VAR_IN_OUT
	rBnt_BlueflagNum: UINT;
	rBnt_Blueflaging: BOOL;	
	NumberPos: ARRAY[0..20] OF LREAL;//接带点记录数据
	NumberPos1: ARRAY[0..20] OF LREAL;//接带点记录数据
	NumberPos2: ARRAY[0..20] OF LREAL;//接带点记录数据
END_VAR

rBnt_Blueflag(CLK:=Bnt_Blueflag , Q=> );	// 接带输入信号
rFlagDone(CLK:=FlagDone , Q=> );	// 电芯下料完成信号
//根据接带信号记录放卷轴当前的角度
IF rBnt_Blueflag.Q THEN
		rBnt_Blueflaging:=TRUE;//接带信号
		rBnt_BlueflagNum:=rBnt_BlueflagCaNum;
		FOR i:=0 TO 20 BY 1 DO
							IF i<20 THEN
									NumberPos[20-i]:=	NumberPos[19-i];
							ELSE
									NumberPos[0]:=AixsoActPos;
							END_IF;
							
							IF i<20 THEN
									NumberPos1[20-i]:=	NumberPos1[19-i];
							ELSE
									NumberPos1[0]:=AixsoActPos+fYDLength;
							END_IF;
							
							IF i<20 THEN
									NumberPos2[20-i]:=	NumberPos2[19-i];
							ELSE
									NumberPos2[0]:=AixsoActPos+fYDLength*2;
							END_IF;
		END_FOR
END_IF
//根据当前的角度
FOR i:=0 TO 20 BY 1 DO
		IF NumberPos[i]<>0 THEN
			RemberPos[i]:= FC_AngleToLength(ABS(AixsoActPos-NumberPos[i]),Diameter);			
		END_IF
		
		IF NumberPos1[i]<>0 THEN
			RemberPos1[i]:= FC_AngleToLength(ABS(AixsoActPos-NumberPos1[i]),Diameter);
		END_IF
		
		IF NumberPos2[i]<>0 THEN
			RemberPos2[i]:= FC_AngleToLength(ABS(AixsoActPos-NumberPos2[i]),Diameter);
		END_IF

		IF (RemberPos[i] >= SetLenght AND NumberPos[i]<>0) OR (RemberPos1[i] >= SetLenght AND NumberPos1[i]<>0)OR (RemberPos2[i] >= SetLenght AND NumberPos2[i]<>0)   THEN
			FlagPoisn[i]:=TRUE;
		END_IF
		
		IF (RemberPos[i] >= SetLenght AND NumberPos[i]<>0) AND rFlagDone.Q THEN
			FlagPoisn[i] :=FALSE;
			NumberPos[i]:=0;
		END_IF
	
		IF (RemberPos1[i] >= SetLenght AND NumberPos1[i]<>0) AND rFlagDone.Q THEN
			FlagPoisn[i] :=FALSE;
			NumberPos1[i]:=0;
		END_IF	

		IF (RemberPos2[i] >= SetLenght AND NumberPos2[i]<>0) AND rFlagDone.Q THEN
			FlagPoisn[i] :=FALSE;
			NumberPos2[i]:=0;
		END_IF		
END_FOR

END_FUNCTION_BLOCK

// ---- P2POUs/BasicFunction/09_User1/FB_CrectCamUpDown_4.TcPOU
FUNCTION_BLOCK FB_CrectCamUpDown_4	
VAR_INPUT
   	bCreatTable		                         :BOOL;	
	Reset                                        :BOOL;  
	iTable		                                :UINT;    

	fInitLength									:REAL;//耦合的初始高度
    fMoveLength                              :REAL;   //目标取或放料高度
    fSaveLength                               :REAL;    //升降安全高度

    fMasterKeyPos1                           :REAL:=208;   
    fMasterKeyPos2                           :REAL:=256;   
END_VAR

VAR_IN_OUT
	axisSlave		                            :axis_ref;  
	axisMaster		                            :axis_ref;  
END_VAR

VAR_OUTPUT
    bCreatTableDone                        :BOOL;
    bCreatTableError                        :BOOL;
	bError                         :BOOL;

END_VAR


VAR
	rtrigs		                                      :ARRAY[1..3]OF R_TRIG;
	ftrigs		                                      :ARRAY[1..3]OF F_TRIG;
    PositionData1			                  :ARRAY[1..8] OF MC_MotionFunctionPoint;	////
	fbCamtableselect:		               	MC_CamTableSelect;////
	Cam_table:				MC_CAM_REF;////
	bWriteCamData: BOOL;
    iCreatTableStep       :INT;
END_VAR


rtrigs[1](CLK:=bCreatTable);  
ftrigs[1](CLK:=bCreatTable);  

CASE iCreatTableStep OF   
0:  
    IF  rtrigs[1].Q  AND NOT bCreatTableError  THEN
         fbCamtableselect.Execute:=FALSE;
         bCreatTableDone:=FALSE;
         bCreatTable:=FALSE;
         bWriteCamData:=TRUE;
         iCreatTableStep:=10;
    END_IF 

10: 
   IF NOT bWriteCamData THEN 
	  fbCamtableselect.Execute:=TRUE;   
	 iCreatTableStep:=20;	
  END_IF

20:		
	IF NOT  fbCamtableselect.Execute   THEN
        bCreatTableDone:=TRUE;
		iCreatTableStep:=0;	
    ELSIF  fbCamtableselect.Error        THEN
       bCreatTableError:=TRUE;
       iCreatTableStep:=999;	//创建凸轮失败
	END_IF		
END_CASE

(**********故障***********)
	IF  Reset  AND bCreatTableError  THEN  
	   bCreatTableError:=FALSE;
	   iCreatTableStep:=0;
	END_IF


ModifyCam();

ACTION ModifyCam:

fbCamtableselect(   
	Execute:=                        fbCamtableselect.Execute ,
	Periodic:=                        FALSE ,
	MasterAbsolute:=             FALSE,
	SlaveAbsolute:=                FALSE ,
	CamTableID:=                  iTable,
	Master:=                         axisMaster ,
	Slave:=                            axisSlave ,
	CamTable:=                     Cam_table , );

IF fbCamtableselect.Done THEN
    fbCamtableselect.Execute:=FALSE;
END_IF

IF bWriteCamData  THEN
 
	  Cam_table.ArraySize:=SIZEOF(PositionData1); 
	  Cam_table.NoOfColumns:=1;
	  Cam_table.NoOfRows:=4;
	  Cam_table.pArray:=ADR(PositionData1);
	  Cam_table.TableType:=MC_TABLETYPE_MOTIONFUNCTION;
  
      //MOTIONFUNCTYPE_BESCHLTRAPEZ     MOTIONFUNCTYPE_POLYNOM7_MM    MOTIONFUNCTYPE_BESCHLTRAPEZ   MOTIONFUNCTYPE_POLYNOM1

	  PositionData1[1].	PointIndex	:=	        1;
	  PositionData1[1].	FunctionType	:=		MOTIONFUNCTYPE_POLYNOM5_MM;//MOTIONFUNCTYPE_BESCHLTRAPEZ     MOTIONFUNCTYPE_POLYNOM7_MM    MOTIONFUNCTYPE_BESCHLTRAPEZ
	  PositionData1[1].	PointType	:=	        MOTIONPOINTTYPE_MOTION;
	  PositionData1[1].	RelIndexNextPoint	:=  1;
	  PositionData1[1].	MasterPos	:=	        0;
	  PositionData1[1].	SlavePos	:=	        0;		//fMoveLength
	  PositionData1[1].	SlaveVelo	:=	        0;
	  
	  PositionData1[2].	PointIndex	:=	        2;
	  PositionData1[2].	FunctionType	:=		MOTIONFUNCTYPE_POLYNOM5_MM;
	  PositionData1[2].	PointType	:=	        MOTIONPOINTTYPE_MOTION;
	  PositionData1[2].	RelIndexNextPoint	:=  1;
	  PositionData1[2].	MasterPos	:=	        fMasterKeyPos1;//fMasterKeyPos
	  PositionData1[2].	SlavePos	:=	        fSaveLength - fInitLength;	
	  PositionData1[2].	SlaveVelo	:=	        0;//(fInitLength-fSaveLength)/fMasterKeyPos1	;

	  PositionData1[3].	PointIndex	:=	        3;//SJ
	  PositionData1[3].	FunctionType	:=		MOTIONFUNCTYPE_POLYNOM1;
	  PositionData1[3].	PointType	:=	        MOTIONPOINTTYPE_MOTION;
	  PositionData1[3].	RelIndexNextPoint	:=  1;
	  PositionData1[3].	MasterPos	:=	        fMasterKeyPos2;//fMasterKeyPos
	  PositionData1[3].	SlavePos	:=	        0;	
	  PositionData1[3].	SlaveVelo	:=	        0;//(fInitLength-fSaveLength)/fMasterKeyPos1	;	  
	  
	  
	  PositionData1[4].	PointIndex	:=	        4;
	  PositionData1[4].	FunctionType	:=		MOTIONFUNCTYPE_POLYNOM5_MM;
	  PositionData1[4].	PointType	:=	        MOTIONPOINTTYPE_MOTION;
	  PositionData1[4].	RelIndexNextPoint	:=  0;
	  PositionData1[4].	MasterPos	:=	        360;//fMasterKeyPos
	  PositionData1[4].	SlavePos	:=	        0;	
	  PositionData1[4].	SlaveVelo	:=	        0;//(fInitLength-fSaveLength)/fMasterKeyPos1	;
	  



     bWriteCamData:=FALSE;
END_IF
END_ACTION

END_FUNCTION_BLOCK

// ---- P2POUs/BasicFunction/12_User2/FB_DiameterORLength.TcPOU
FUNCTION_BLOCK FB_DiameterORLength
VAR_INPUT
	D1 : REAL; //外直径
	R1 : REAL:=172; //内直径
	T1 : REAL; //隔膜厚度
END_VAR
VAR_OUTPUT
	OUT1: REAL;
END_VAR
VAR
	R2: REAL;
	R3: REAL;
	R4: REAL;
	
END_VAR

IF  T1 <> 0 AND D1 >= R1 THEN
	R2:=(D1-R1)/2  ;  
	R3:=((D1*Tc2_System.PI)+(R1*Tc2_System.PI))/2 ;  //平均长度
	R4:=R2/T1;  //总层数
	OUT1:=(R4*R3)/1000;
END_IF

END_FUNCTION_BLOCK

// ---- P2POUs/BasicFunction/12_User2/FB_RectifyTry.TcPOU
FUNCTION_BLOCK FB_RectifyTry
VAR_INPUT
	Execute: BOOL;// 测试启动HMI
	AxisNO_X: INT; // X轴	
	AxisNO_Y: INT; // Y轴	
	AxisNO_R: INT; // R轴	
	Demarcate_X:REAL;//X轴纠偏位
	Demarcate_Y:REAL;//Y轴纠偏位	
	Demarcate_R:REAL;//R轴纠偏位		
	// CCD拍照记录次数
	CCDNo: INT;
END_VAR
VAR_OUTPUT
END_VAR
VAR
	Step0: INT;
	r_TRIG: R_TRIG;

	// 延时复位CCD拍照启动
	TON1: TON;
	TON2: TON;
	i: INT;
END_VAR

VAR_IN_OUT
	// 启动CCD拍照
	CCDStart: BOOL;
END_VAR

//纠偏平台定位精度数据测试
r_TRIG(CLK:=Execute , Q=> );
TON1(IN:= , PT:=T#2S , Q=> , ET=> );
TON2(IN:= , PT:=T#0.3S , Q=> , ET=> );

CASE Step0 OF
	0://判断是否启动测试
		IF r_TRIG.Q THEN
			i:=0;
			Step0:=10;
			TON2.IN:=FALSE;
		END_IF
	10://纠偏平台X、Y回初始位
		IF arrAxisCtrl[AxisNO_X].Status.Homed AND arrAxisCtrl[AxisNO_X].Status.NoMoving THEN
				IF arrAxisCtrl[AxisNO_X].Cmd.arrbRealPoint[1] THEN
					arrAxisCtrl[AxisNO_X].Cmd.iGoSetPos:=0;
				ELSE
					arrAxisCtrl[AxisNO_X].Cmd.iGoSetPos:=1;
				END_IF
		END_IF
		IF arrAxisCtrl[AxisNO_Y].Status.Homed AND arrAxisCtrl[AxisNO_Y].Status.NoMoving  THEN
				IF arrAxisCtrl[AxisNO_Y].Cmd.arrbRealPoint[1] THEN
					arrAxisCtrl[AxisNO_Y].Cmd.iGoSetPos:=0;
				ELSE
					arrAxisCtrl[AxisNO_Y].Cmd.iGoSetPos:=1;
				END_IF
		END_IF	
	  IF arrAxisCtrl[AxisNO_R].Status.Homed AND arrAxisCtrl[AxisNO_R].Status.NoMoving  THEN
			IF arrAxisCtrl[AxisNO_R].Cmd.arrbRealPoint[1] THEN
				arrAxisCtrl[AxisNO_R].Cmd.iGoSetPos:=0;							       
			ELSE
				arrAxisCtrl[AxisNO_R].Cmd.iGoSetPos:=1;
			END_IF
		END_IF		
		
		IF  arrAxisCtrl[AxisNO_X].Cmd.arrbRealPoint[1]  AND arrAxisCtrl[AxisNO_Y].Cmd.arrbRealPoint[1]  AND arrAxisCtrl[AxisNO_R].Cmd.arrbRealPoint[1] AND
			 arrAxisCtrl[AxisNO_X].Status.Homed AND  arrAxisCtrl[AxisNO_Y].Status.Homed AND arrAxisCtrl[AxisNO_R].Status.Homed THEN
				Step0:=30;
				TON2.IN:=TRUE;
		END_IF	
	(*20://纠偏平台R回初始位
		IF arrAxisCtrl[AxisNO_R].Status.Homed AND arrAxisCtrl[AxisNO_R].Status.NoMoving  THEN
			IF arrAxisCtrl[AxisNO_R].Cmd.arrbRealPoint[1] THEN
				arrAxisCtrl[AxisNO_R].Cmd.iGoSetPos:=0;
				Step0:=30;									       
			ELSE
				arrAxisCtrl[AxisNO_R].Cmd.iGoSetPos:=1;
			END_IF
		END_IF*)
	30://启动CCD拍照
	  IF TON2.Q THEN
		CCDStart:=TRUE;   //CCD拍照启动
		TON2.IN:=FALSE;
		Step0:=40;
	  END_IF	
	40://延时复位CDD拍照启动信号
		IF NOT TON1.Q THEN
			TON1.IN:=TRUE;
		ELSE
			CCDStart:=FALSE;   //CCD拍照启动
			TON1.IN:=FALSE;
			Step0:=50;
		END_IF
	50://纠偏平台X、Y纠偏量
		arrAxisPar[AxisNO_X].arrTargetPoint[6]:=arrAxisPar[AxisNO_X].arrTargetPoint[1] + Demarcate_X;
		arrAxisPar[AxisNO_Y].arrTargetPoint[6]:=arrAxisPar[AxisNO_Y].arrTargetPoint[1] + Demarcate_Y;
		arrAxisPar[AxisNO_R].arrTargetPoint[6]:=arrAxisPar[AxisNO_R].arrTargetPoint[1] +Demarcate_R;
		Step0:=60;	
		TON2.IN:=FALSE;
	60://纠偏平台X、Y移动至纠偏位
 		IF arrAxisCtrl[AxisNO_X].Status.Homed AND arrAxisCtrl[AxisNO_X].Status.NoMoving THEN
				IF arrAxisCtrl[AxisNO_X].Cmd.arrbRealPoint[6] THEN
					arrAxisCtrl[AxisNO_X].Cmd.iGoSetPos:=0;
				ELSE
					arrAxisCtrl[AxisNO_X].Cmd.iGoSetPos:=6;
				END_IF
		END_IF
		IF arrAxisCtrl[AxisNO_Y].Status.Homed AND arrAxisCtrl[AxisNO_Y].Status.NoMoving  THEN
				IF arrAxisCtrl[AxisNO_Y].Cmd.arrbRealPoint[6] THEN
					arrAxisCtrl[AxisNO_Y].Cmd.iGoSetPos:=0;
				ELSE
					arrAxisCtrl[AxisNO_Y].Cmd.iGoSetPos:=6;
				END_IF
		END_IF	
		
	 	IF arrAxisCtrl[AxisNO_R].Status.Homed AND arrAxisCtrl[AxisNO_R].Status.NoMoving THEN
				IF arrAxisCtrl[AxisNO_R].Cmd.arrbRealPoint[6] THEN
					arrAxisCtrl[AxisNO_R].Cmd.iGoSetPos:=0;
				ELSE
					arrAxisCtrl[AxisNO_R].Cmd.iGoSetPos:=6;
				END_IF
		END_IF
	
		IF  arrAxisCtrl[AxisNO_X].Cmd.arrbRealPoint[6]  AND arrAxisCtrl[AxisNO_Y].Cmd.arrbRealPoint[6] AND arrAxisCtrl[AxisNO_R].Cmd.arrbRealPoint[6]  AND 
			 arrAxisCtrl[AxisNO_X].Status.Homed AND  arrAxisCtrl[AxisNO_Y].Status.Homed AND  arrAxisCtrl[AxisNO_R].Status.Homed  THEN
			 Step0:=90;
			 TON2.IN:=TRUE;
		END_IF	 
	(*	
	70://纠偏平台R纠偏量
		arrAxisPar[AxisNO_R].arrTargetPoint[4]:=arrAxisPar[AxisNO_R].arrTargetPoint[1] +Demarcate_R;//arrAxisPar[AxisNO_R].arrTargetPoint[1] + 80*SIN(DEG_TO_RAD(Demarcate_R)) ;
		Step0:=80;
	80://纠偏平台R移动到纠偏位
 		IF arrAxisCtrl[AxisNO_R].Status.Homed AND arrAxisCtrl[AxisNO_R].Status.NoMoving THEN
				IF arrAxisCtrl[AxisNO_R].Cmd.arrbRealPoint[4] THEN
					arrAxisCtrl[AxisNO_R].Cmd.iGoSetPos:=0;
				ELSE
					arrAxisCtrl[AxisNO_R].Cmd.iGoSetPos:=4;
				END_IF
		END_IF
		IF  arrAxisCtrl[AxisNO_R].Cmd.arrbRealPoint[4]  AND arrAxisCtrl[AxisNO_R].Status.Homed THEN
			 Step0:=90;
		END_IF	 *)
	90://启动CCD拍照
	IF TON2.Q THEN
		CCDStart:=TRUE;   //CCD拍照启动
		i:=i+1;
		Step0:=100;
		 TON2.IN:=FALSE;
	END_IF		
	100://延时复位CDD拍照启动信号
		IF NOT TON1.Q THEN
			TON1.IN:=TRUE;
		ELSE
			CCDStart:=FALSE;   //CCD拍照启动
			TON1.IN:=FALSE;
			Step0:=110;
		END_IF
	110://判断是否达到设定次数
		IF i>=CCDNo THEN
			i:=0;
			Step0:=0;
		ELSE
			Step0:=10;
		END_IF
END_CASE

END_FUNCTION_BLOCK

// ---- P2POUs/BasicFunction/12_User2/FB_SuckerTest.TcPOU
FUNCTION_BLOCK FB_SuckerTest
VAR_INPUT
	Execute: BOOL;// 测试启动HMI
	AxisNO_1: INT; // 升降轴
	AxisNO_2: INT;//平移轴
	AxisNO_X: INT; // X轴	
	AxisNO_Y: INT; // Y轴	
	AxisNO_R: INT; // R轴	
	CCD_X1:REAL;//CCD拍照X轴方向的纠偏值
	CCD_X2:REAL;//CCD拍照Y轴方的纠偏值
	CCD_Y:REAL;//CCD拍照旋转方向的纠偏值	
	DTCarryingVacuum: INT;//叠台真空
	deviationVacuum: INT;//纠偏平台真空
	deviationVacuumBark: INT;//纠偏平台破真空
	CCDCount: INT;//测试次数
	DTiMode: INT;
END_VAR
VAR_OUTPUT
END_VAR
VAR
	Step0: INT;
	i: INT;
	r_TRIG:R_TRIG;
	TON1: TON;
	TON2: TON;
	TON3: TON;
	TON4: TON;
END_VAR
VAR_IN_OUT
	// 启动CCD拍照
	CCDStart: BOOL;
END_VAR

r_TRIG(CLK:=Execute , Q=> );
TON1(IN:= , PT:=T#0.5S , Q=> , ET=> );
TON2(IN:= , PT:=T#0.3S , Q=> , ET=> );
TON3(IN:= , PT:=T#0.3S , Q=> , ET=> );
TON4(IN:= , PT:=T#0.3S , Q=> , ET=> );
IF DTiMode=3 THEN
CASE Step0 OF
	0://判断是否启动测试
		IF r_TRIG.Q THEN
			i:=0;
			Step0:=10;
			TON2.IN:=FALSE;
		END_IF
	10://纠偏平台X、Y、R 回初始位 、叠台升降去等待高度、
	   IF arrAxisCtrl[AxisNO_1].Status.Homed AND arrAxisCtrl[AxisNO_1].Status.NoMoving THEN
				IF arrAxisCtrl[AxisNO_1].Cmd.arrbRealPoint[4] THEN
					arrAxisCtrl[AxisNO_1].Cmd.iGoSetPos:=0;
				ELSE
					arrAxisCtrl[AxisNO_1].Cmd.iGoSetPos:=4;
				END_IF
		END_IF
		
		IF arrAxisCtrl[AxisNO_X].Status.Homed AND arrAxisCtrl[AxisNO_X].Status.NoMoving THEN
				IF arrAxisCtrl[AxisNO_X].Cmd.arrbRealPoint[1] THEN
					arrAxisCtrl[AxisNO_X].Cmd.iGoSetPos:=0;
				ELSE
					arrAxisCtrl[AxisNO_X].Cmd.iGoSetPos:=1;
				END_IF
		END_IF
		IF arrAxisCtrl[AxisNO_Y].Status.Homed AND arrAxisCtrl[AxisNO_Y].Status.NoMoving  THEN
				IF arrAxisCtrl[AxisNO_Y].Cmd.arrbRealPoint[1] THEN
					arrAxisCtrl[AxisNO_Y].Cmd.iGoSetPos:=0;
				ELSE
					arrAxisCtrl[AxisNO_Y].Cmd.iGoSetPos:=1;
				END_IF
		END_IF	
	  IF arrAxisCtrl[AxisNO_R].Status.Homed AND arrAxisCtrl[AxisNO_R].Status.NoMoving  THEN
			IF arrAxisCtrl[AxisNO_R].Cmd.arrbRealPoint[1] THEN
				arrAxisCtrl[AxisNO_R].Cmd.iGoSetPos:=0;							       
			ELSE
				arrAxisCtrl[AxisNO_R].Cmd.iGoSetPos:=1;
			END_IF
		END_IF		
		
		IF  arrAxisCtrl[AxisNO_X].Cmd.arrbRealPoint[1]  AND arrAxisCtrl[AxisNO_Y].Cmd.arrbRealPoint[1]  AND arrAxisCtrl[AxisNO_R].Cmd.arrbRealPoint[1] AND
		    arrAxisCtrl[AxisNO_1].Status.NoMoving AND arrAxisCtrl[AxisNO_X].Status.NoMoving AND arrAxisCtrl[AxisNO_Y].Status.NoMoving AND arrAxisCtrl[AxisNO_R].Status.NoMoving AND 
		    arrAxisCtrl[AxisNO_1].Cmd.arrbRealPoint[4] THEN
		  Step0:=20;
		END_IF
	20://叠台升降去取片位
		IF arrAxisCtrl[AxisNO_1].Status.Homed AND arrAxisCtrl[AxisNO_1].Status.NoMoving  AND  arrAxisCtrl[AxisNO_2].Cmd.arrbRealPoint[1] THEN
				IF arrAxisCtrl[AxisNO_1].Cmd.arrbRealPoint[2] THEN
					arrAxisCtrl[AxisNO_1].Cmd.iGoSetPos:=0;
				TON3.IN:=FALSE;
				Step0:=30;					
				ELSE
					arrAxisCtrl[AxisNO_1].Cmd.iGoSetPos:=2;
				END_IF
				
		END_IF
	30://叠台升降开真空、纠偏平台破真空
	        arrCyCtrl[DTCarryingVacuum].Cmd.bON:=FALSE;//叠片搬运升降真空开
			arrCyCtrl[DTCarryingVacuum].Cmd.bOFF:=TRUE;//叠片搬运升降真空开
	   	IF arrAxisCtrl[AxisNO_1].Status.Homed AND arrAxisCtrl[AxisNO_1].Status.NoMoving AND NOT arrAxisCtrl[AxisNO_1].Status.Error AND
				arrAxisCtrl[AxisNO_1].Cmd.arrbRealPoint[2] THEN
					arrCyCtrl[deviationVacuum].Cmd.bOFF:=TRUE;//纠偏平台真空关闭
					arrCyCtrl[deviationVacuum].Cmd.bON:=FALSE;//纠偏平台真空关闭
					arrCyCtrl[deviationVacuumBark].Cmd.bON:=TRUE;//纠偏平台破真空打开	
					arrCyCtrl[deviationVacuumBark].Cmd.bOFF:=FALSE;//纠偏平台破真空打开       
	                       IF NOT TON3.Q THEN
			                  TON3.IN:=TRUE;
				           ELSE
					          TON3.IN:=FALSE;
							  TON4.IN:=FALSE;
                               Step0:=31;
                           END_IF           	
		END_IF
		
     31://叠台升降去等待高度
	 
        IF arrAxisCtrl[AxisNO_1].Status.Homed AND arrAxisCtrl[AxisNO_1].Status.NoMoving THEN
				IF arrAxisCtrl[AxisNO_1].Cmd.arrbRealPoint[4] THEN
					arrAxisCtrl[AxisNO_1].Cmd.iGoSetPos:=0;
					Step0:=32;
				   TON4.IN:=TRUE;
				ELSE
					arrAxisCtrl[AxisNO_1].Cmd.iGoSetPos:=4;
				END_IF
			
		END_IF

	32://叠台升降去放片位
	    IF arrAxisCtrl[AxisNO_1].Status.Homed AND arrAxisCtrl[AxisNO_1].Status.NoMoving  AND  arrAxisCtrl[AxisNO_2].Cmd.arrbRealPoint[1] AND TON4.Q  THEN
				IF arrAxisCtrl[AxisNO_1].Cmd.arrbRealPoint[2] THEN
					arrAxisCtrl[AxisNO_1].Cmd.iGoSetPos:=0;
					Step0:=33;
					TON4.IN:=FALSE;
				ELSE
					arrAxisCtrl[AxisNO_1].Cmd.iGoSetPos:=2;
				END_IF
				
				
		END_IF
	33://叠台升降开破真空、纠偏平台真空
	IF arrAxisCtrl[AxisNO_1].Status.Homed AND arrAxisCtrl[AxisNO_1].Status.NoMoving AND NOT arrAxisCtrl[AxisNO_1].Status.Error AND
       arrAxisCtrl[AxisNO_1].Cmd.arrbRealPoint[2] THEN
				  arrCyCtrl[DTCarryingVacuum].Cmd.bON:=TRUE;//叠片搬运升降破真空开
				  arrCyCtrl[DTCarryingVacuum].Cmd.bOFF:=FALSE;//叠片搬运升降破真空开
				  arrCyCtrl[deviationVacuum].Cmd.bOFF:=FALSE;//纠偏平台真空打开
				  arrCyCtrl[deviationVacuum].Cmd.bON:=TRUE;//纠偏平台真空打开 
			      TON2.IN:=TRUE;
			      Step0:=40;
	END_IF
	40://启动CCD拍照
	IF TON2.Q THEN
		TON2.IN:=FALSE;
		Step0:=50;
	  END_IF	

	50://叠台升降去等待高度
		IF arrAxisCtrl[AxisNO_1].Status.Homed AND arrAxisCtrl[AxisNO_1].Status.NoMoving THEN
			IF arrAxisCtrl[AxisNO_1].Cmd.arrbRealPoint[4] THEN
					arrAxisCtrl[AxisNO_1].Cmd.iGoSetPos:=0;
					 Step0:=60;
					 CCDStart:=TRUE;   //CCD拍照启动
				ELSE
					arrAxisCtrl[AxisNO_1].Cmd.iGoSetPos:=4;
				END_IF
		END_IF
	 60://延时复位CDD拍照启动信号
		IF NOT TON1.Q THEN
			TON1.IN:=TRUE;
		ELSE
			CCDStart:=FALSE;   //CCD拍照启动
			TON1.IN:=FALSE;
			Step0:=65;
		END_IF
	
    65:
			arrAxisPar[AxisNO_X].arrTargetPoint[2]:=arrAxisPar[AxisNO_X].arrTargetPoint[1]+CCD_X1;//+(103.94*COS(DEG_TO_RAD(CCD_W+225))-103.94*COS(DEG_TO_RAD(225))); 
			arrAxisPar[AxisNO_Y].arrTargetPoint[2]:=arrAxisPar[AxisNO_Y].arrTargetPoint[1]+CCD_X2;//+(103.94*SIN(DEG_TO_RAD(CCD_W+315))-103.94*COS(DEG_TO_RAD(315)));
			arrAxisPar[AxisNO_R].arrTargetPoint[2]:=arrAxisPar[AxisNO_R].arrTargetPoint[1]+CCD_Y;//+(103.94*COS(DEG_TO_RAD(CCD_W+135))-103.94*COS(DEG_TO_RAD(135)));	
			Step0:=70;
			
	70://纠偏平台X、Y、R去纠偏位
		IF arrAxisCtrl[AxisNO_X].Status.Homed AND arrAxisCtrl[AxisNO_X].Status.NoMoving THEN
				IF arrAxisCtrl[AxisNO_X].Cmd.arrbRealPoint[2] THEN
					arrAxisCtrl[AxisNO_X].Cmd.iGoSetPos:=0;
				ELSE
					arrAxisCtrl[AxisNO_X].Cmd.iGoSetPos:=2;
				END_IF
		END_IF
		IF arrAxisCtrl[AxisNO_Y].Status.Homed AND arrAxisCtrl[AxisNO_Y].Status.NoMoving  THEN
				IF arrAxisCtrl[AxisNO_Y].Cmd.arrbRealPoint[2] THEN
					arrAxisCtrl[AxisNO_Y].Cmd.iGoSetPos:=0;
				ELSE
					arrAxisCtrl[AxisNO_Y].Cmd.iGoSetPos:=2;
				END_IF
		END_IF	
	  IF arrAxisCtrl[AxisNO_R].Status.Homed AND arrAxisCtrl[AxisNO_R].Status.NoMoving  THEN
			IF arrAxisCtrl[AxisNO_R].Cmd.arrbRealPoint[2] THEN
				arrAxisCtrl[AxisNO_R].Cmd.iGoSetPos:=0;							       
			ELSE
				arrAxisCtrl[AxisNO_R].Cmd.iGoSetPos:=2;
			END_IF
		END_IF		

		IF  arrAxisCtrl[AxisNO_X].Cmd.arrbRealPoint[2]  AND arrAxisCtrl[AxisNO_Y].Cmd.arrbRealPoint[2]  AND arrAxisCtrl[AxisNO_R].Cmd.arrbRealPoint[2] AND
		    arrAxisCtrl[AxisNO_X].Status.NoMoving AND arrAxisCtrl[AxisNO_Y].Status.NoMoving AND arrAxisCtrl[AxisNO_R].Status.NoMoving THEN
			 TON2.IN:=TRUE;
			  Step0:=90;
	   END_IF
	90://启动CCD拍照
	IF TON2.Q THEN
		CCDStart:=TRUE;   //CCD拍照启动
		i:=i+1;
		Step0:=100;
		 TON2.IN:=FALSE;
	END_IF		
	100://延时复位CDD拍照启动信号
		IF NOT TON1.Q THEN
			TON1.IN:=TRUE;
		ELSE
			CCDStart:=FALSE;   //CCD拍照启动
			TON1.IN:=FALSE;
			Step0:=110;
		END_IF
	110://纠偏平台X、Y、R 回初始位 
	IF arrAxisCtrl[AxisNO_X].Status.Homed AND arrAxisCtrl[AxisNO_X].Status.NoMoving THEN
				IF arrAxisCtrl[AxisNO_X].Cmd.arrbRealPoint[1] THEN
					arrAxisCtrl[AxisNO_X].Cmd.iGoSetPos:=0;
				ELSE
					arrAxisCtrl[AxisNO_X].Cmd.iGoSetPos:=1;
				END_IF
		END_IF
		IF arrAxisCtrl[AxisNO_Y].Status.Homed AND arrAxisCtrl[AxisNO_Y].Status.NoMoving  THEN
				IF arrAxisCtrl[AxisNO_Y].Cmd.arrbRealPoint[1] THEN
					arrAxisCtrl[AxisNO_Y].Cmd.iGoSetPos:=0;
				ELSE
					arrAxisCtrl[AxisNO_Y].Cmd.iGoSetPos:=1;
				END_IF
		END_IF	
	  IF arrAxisCtrl[AxisNO_R].Status.Homed AND arrAxisCtrl[AxisNO_R].Status.NoMoving  THEN
			IF arrAxisCtrl[AxisNO_R].Cmd.arrbRealPoint[1] THEN
				arrAxisCtrl[AxisNO_R].Cmd.iGoSetPos:=0;							       
			ELSE
				arrAxisCtrl[AxisNO_R].Cmd.iGoSetPos:=1;
			END_IF
		END_IF	
	   IF  arrAxisCtrl[AxisNO_X].Cmd.arrbRealPoint[1]  AND arrAxisCtrl[AxisNO_Y].Cmd.arrbRealPoint[1]  AND arrAxisCtrl[AxisNO_R].Cmd.arrbRealPoint[1] AND
		   arrAxisCtrl[AxisNO_X].Status.NoMoving AND arrAxisCtrl[AxisNO_Y].Status.NoMoving AND arrAxisCtrl[AxisNO_R].Status.NoMoving THEN
				                    Step0:=120;
		END_IF	
	120://判断是否达到设定次数
		IF i>=CCDCount THEN
			i:=0;
			Step0:=0;
		ELSE
			Step0:=10;
		END_IF
END_CASE
END_IF

END_FUNCTION_BLOCK

// ---- P2POUs/BasicFunction/09_User1/FB_CrectCamYaDaoLine2_V2.TcPOU
FUNCTION_BLOCK FB_CrectCamYaDaoLine2_V2	
VAR_INPUT
   	bCreatTable		                         :BOOL;	
	Reset                                        :BOOL;  
	iTable		                                :UINT;    


    fMoveLength                                 :REAL:=40;   //压倒平移最大距离
    
    fMasterKeyPos1                           :REAL:=164;   
    fMasterKeyPos2                           :REAL:=241;   
    fMasterKeyPos3                           :REAL:=289;  
    fMasterKeyPos4                           :REAL:=289;  
	 
	fMoveLength2                             :REAL:=-15;   //压刀压隔膜长度
END_VAR

VAR_IN_OUT
	axisSlave		                            :axis_ref;  
	axisMaster		                            :axis_ref;  
END_VAR

VAR_OUTPUT
    bCreatTableDone                        :BOOL;
    bCreatTableError                        :BOOL;
	bError                         :BOOL;

END_VAR


VAR
	rtrigs		                                      :ARRAY[1..3]OF R_TRIG;
	ftrigs		                                      :ARRAY[1..3]OF F_TRIG;
    PositionData1			                  :ARRAY[1..6] OF MC_MotionFunctionPoint;	////
	fbCamtableselect:		               	MC_CamTableSelect;////
	Cam_table:				MC_CAM_REF;////
	bWriteCamData: BOOL;
    iCreatTableStep       :INT;
END_VAR


rtrigs[1](CLK:=bCreatTable);  
ftrigs[1](CLK:=bCreatTable);  

CASE iCreatTableStep OF   
0:  
    IF  rtrigs[1].Q  AND NOT bCreatTableError  THEN
         fbCamtableselect.Execute:=FALSE;
         bCreatTableDone:=FALSE;
         bCreatTable:=FALSE;
         bWriteCamData:=TRUE;
         iCreatTableStep:=10;
    END_IF 

10: 
   IF NOT bWriteCamData THEN 
	  fbCamtableselect.Execute:=TRUE;   
	 iCreatTableStep:=20;	
  END_IF

20:		
	IF NOT  fbCamtableselect.Execute   THEN
        bCreatTableDone:=TRUE;
		iCreatTableStep:=0;	
    ELSIF  fbCamtableselect.Error        THEN
       bCreatTableError:=TRUE;
       iCreatTableStep:=999;	//创建凸轮失败
	END_IF		
END_CASE

(**********故障***********)
	IF  Reset  AND bCreatTableError  THEN  
	   bCreatTableError:=FALSE;
	   iCreatTableStep:=0;
	END_IF


ModifyCam();

ACTION ModifyCam:

fbCamtableselect(   
	Execute:=                        fbCamtableselect.Execute ,
	Periodic:=                        FALSE ,
	MasterAbsolute:=             FALSE,
	SlaveAbsolute:=                FALSE ,
	CamTableID:=                  iTable,
	Master:=                         axisMaster ,
	Slave:=                            axisSlave ,
	CamTable:=                     Cam_table , );

IF fbCamtableselect.Done THEN
    fbCamtableselect.Execute:=FALSE;
END_IF

IF bWriteCamData  THEN

	  Cam_table.ArraySize:=SIZEOF(PositionData1); 
	  Cam_table.NoOfColumns:=1;
	  Cam_table.NoOfRows:=4;
	  Cam_table.pArray:=ADR(PositionData1);
	  Cam_table.TableType:=MC_TABLETYPE_MOTIONFUNCTION;
  
      //MOTIONFUNCTYPE_BESCHLTRAPEZ     MOTIONFUNCTYPE_POLYNOM7_MM    MOTIONFUNCTYPE_BESCHLTRAPEZ   MOTIONFUNCTYPE_POLYNOM1

	  PositionData1[1].	PointIndex	:=	        1;
	  PositionData1[1].	FunctionType	:=		MOTIONFUNCTYPE_POLYNOM1;
	  PositionData1[1].	PointType	:=	        MOTIONPOINTTYPE_MOTION;
	  PositionData1[1].	RelIndexNextPoint	:=  1;
	  PositionData1[1].	MasterPos	:=	        0;
	  PositionData1[1].	SlavePos	:=	        0;		//fMoveLength
	  PositionData1[1].	SlaveVelo	:=	        0;
	  
	  PositionData1[2].	PointIndex	:=	        2;
	  PositionData1[2].	FunctionType	:=		MOTIONFUNCTYPE_POLYNOM5_MM;
	  PositionData1[2].	PointType	:=	        MOTIONPOINTTYPE_MOTION;
	  PositionData1[2].	RelIndexNextPoint	:=  1;
	  PositionData1[2].	MasterPos	:=	        fMasterKeyPos1;
	  PositionData1[2].	SlavePos	:=	        0;	
	  PositionData1[2].	SlaveVelo	:=	        0	;
(*
	  PositionData1[3].	PointIndex	:=	        3;
	  PositionData1[3].	FunctionType	:=		MOTIONFUNCTYPE_POLYNOM5_MM;
	  PositionData1[3].	PointType	:=	        MOTIONPOINTTYPE_MOTION;
	  PositionData1[3].	RelIndexNextPoint	:=  0;
	  PositionData1[3].	MasterPos	:=	        fMasterKeyPos2;
	  PositionData1[3].	SlavePos	:=	        fMoveLength;	
	  PositionData1[3].	SlaveVelo	:=	        0	;
*)
	  PositionData1[3].	PointIndex	:=	        3;
	  PositionData1[3].	FunctionType	:=		MOTIONFUNCTYPE_POLYNOM1;
	  PositionData1[3].	PointType	:=	        MOTIONPOINTTYPE_MOTION;
	  PositionData1[3].	RelIndexNextPoint	:=  1;
	  PositionData1[3].	MasterPos	:=	        fMasterKeyPos3;//fMasterKeyPos
	  PositionData1[3].	SlavePos	:=	        fMoveLength;	
	  PositionData1[3].	SlaveVelo	:=	       0	;

	  PositionData1[4].	PointIndex	:=	        4;
	  PositionData1[4].	FunctionType	:=		MOTIONFUNCTYPE_POLYNOM1;
	  PositionData1[4].	PointType	:=	        MOTIONPOINTTYPE_MOTION;
	  PositionData1[4].	RelIndexNextPoint	:=  0;
	  PositionData1[4].	MasterPos	:=	        360;
	  PositionData1[4].	SlavePos	:=	       fMoveLength;	
	  PositionData1[4].	SlaveVelo	:=	       0	;

     bWriteCamData:=FALSE;
END_IF
END_ACTION

END_FUNCTION_BLOCK

// ---- P2POUs/BasicFunction/09_User1/FB_CrectCamYaDaoUpDown2.TcPOU
FUNCTION_BLOCK FB_CrectCamYaDaoUpDown2	
VAR_INPUT
   	bCreatTable		                         :BOOL;	
	Reset                                        :BOOL;  
	iTable		                                :UINT;    

    fMoveLength                              :REAL:=8;   //升降最大距离
    fSaveLength1                               :REAL:=2 ;    //压针抬升高度
    fSaveLength2                               :REAL:=3;  //压针下压高度

    fMasterKeyPos1                           :REAL:=144;   
    fMasterKeyPos2                           :REAL:=164;   
    fMasterKeyPos3                           :REAL:=204;   

    fMasterKeyPos4                           :REAL:=246;   
    fMasterKeyPos5                          :REAL:=289;   
    fMasterKeyPos6                           :REAL:=328;   


END_VAR

VAR_IN_OUT
	axisSlave		                            :axis_ref;  
	axisMaster		                            :axis_ref;  
END_VAR

VAR_OUTPUT
    bCreatTableDone                        :BOOL;
    bCreatTableError                        :BOOL;
	bError                         :BOOL;

END_VAR


VAR
	rtrigs		                                      :ARRAY[1..3]OF R_TRIG;
	ftrigs		                                      :ARRAY[1..3]OF F_TRIG;
    PositionData1			                  :ARRAY[1..8] OF MC_MotionFunctionPoint;	////
	fbCamtableselect:		               	MC_CamTableSelect;////
	Cam_table:				MC_CAM_REF;////
	bWriteCamData: BOOL;
    iCreatTableStep       :INT;
END_VAR


rtrigs[1](CLK:=bCreatTable);  
ftrigs[1](CLK:=bCreatTable);  

CASE iCreatTableStep OF   
0:  
    IF  rtrigs[1].Q  AND NOT bCreatTableError  THEN
         fbCamtableselect.Execute:=FALSE;
         bCreatTableDone:=FALSE;
         bCreatTable:=FALSE;
         bWriteCamData:=TRUE;
         iCreatTableStep:=10;
    END_IF 

10: 
   IF NOT bWriteCamData THEN 
	  fbCamtableselect.Execute:=TRUE;   
	 iCreatTableStep:=20;	
  END_IF

20:		
	IF NOT  fbCamtableselect.Execute   THEN
        bCreatTableDone:=TRUE;
		iCreatTableStep:=0;	
    ELSIF  fbCamtableselect.Error        THEN
       bCreatTableError:=TRUE;
       iCreatTableStep:=999;	//创建凸轮失败
	END_IF		
END_CASE

(**********故障***********)
	IF  Reset  AND bCreatTableError  THEN  
	   bCreatTableError:=FALSE;
	   iCreatTableStep:=0;
	END_IF


ModifyCam();

ACTION ModifyCam:

fbCamtableselect(   
	Execute:=                        fbCamtableselect.Execute ,
	Periodic:=                        FALSE ,
	MasterAbsolute:=             FALSE,
	SlaveAbsolute:=                FALSE ,
	CamTableID:=                  iTable,
	Master:=                         axisMaster ,
	Slave:=                            axisSlave ,
	CamTable:=                     Cam_table , );

IF fbCamtableselect.Done THEN
    fbCamtableselect.Execute:=FALSE;
END_IF

IF bWriteCamData  THEN
 
	  Cam_table.ArraySize:=SIZEOF(PositionData1); 
	  Cam_table.NoOfColumns:=1;
	  Cam_table.NoOfRows:=7;
	  Cam_table.pArray:=ADR(PositionData1);
	  Cam_table.TableType:=MC_TABLETYPE_MOTIONFUNCTION;
      //MOTIONFUNCTYPE_BESCHLTRAPEZ     MOTIONFUNCTYPE_POLYNOM7_MM    MOTIONFUNCTYPE_BESCHLTRAPEZ   MOTIONFUNCTYPE_POLYNOM1

	  PositionData1[1].	PointIndex	:=	        1;
	  PositionData1[1].	FunctionType	:=		MOTIONFUNCTYPE_POLYNOM1;//
	  PositionData1[1].	PointType	:=	        MOTIONPOINTTYPE_MOTION;
	  PositionData1[1].	RelIndexNextPoint	:=  1;
	  PositionData1[1].	MasterPos	:=	        0;
	  PositionData1[1].	SlavePos	:=	        0;		//fMoveLength
	  PositionData1[1].	SlaveVelo	:=	        0;
	  
	  PositionData1[2].	PointIndex	:=	        2;
	  PositionData1[2].	FunctionType	:=		MOTIONFUNCTYPE_POLYNOM5_MM;
	  PositionData1[2].	PointType	:=	        MOTIONPOINTTYPE_MOTION;
	  PositionData1[2].	RelIndexNextPoint	:=  1;
	  PositionData1[2].	MasterPos	:=	        fMasterKeyPos1;
	  PositionData1[2].	SlavePos	:=	        0;	
	  PositionData1[2].	SlaveVelo	:=	       0	;

	  PositionData1[3].	PointIndex	:=	        3;
	  PositionData1[3].	FunctionType	:=		MOTIONFUNCTYPE_POLYNOM1;
	  PositionData1[3].	PointType	:=	        MOTIONPOINTTYPE_MOTION;
	  PositionData1[3].	RelIndexNextPoint	:=  0;
	  PositionData1[3].	MasterPos	:=	        fMasterKeyPos2;
	  PositionData1[3].	SlavePos	:=	        fSaveLength1;	
	  PositionData1[3].	SlaveVelo	:=	        0	;

	  PositionData1[4].	PointIndex	:=	        4;
	  PositionData1[4].	FunctionType	:=		MOTIONFUNCTYPE_POLYNOM5_MM;
	  PositionData1[4].	PointType	:=	        MOTIONPOINTTYPE_MOTION;
	  PositionData1[4].	RelIndexNextPoint	:=  1;
	  PositionData1[4].	MasterPos	:=	        fMasterKeyPos3;
	  PositionData1[4].	SlavePos	:=	        fSaveLength1;	
	  PositionData1[4].	SlaveVelo	:=	       0	;

	  PositionData1[5].	PointIndex	:=	        5;
	  PositionData1[5].	FunctionType	:=		MOTIONFUNCTYPE_POLYNOM5_MM;
	  PositionData1[5].	PointType	:=	        MOTIONPOINTTYPE_MOTION;
	  PositionData1[5].	RelIndexNextPoint	:=  1;
	  PositionData1[5].	MasterPos	:=	        fMasterKeyPos4;
	  PositionData1[5].	SlavePos	:=	        fMoveLength;	
	  PositionData1[5].	SlaveVelo	:=	       0	;
(*
	  PositionData1[6].	PointIndex	:=	        6;
	  PositionData1[6].	FunctionType	:=		MOTIONFUNCTYPE_POLYNOM7_MM;
	  PositionData1[6].	PointType	:=	        MOTIONPOINTTYPE_MOTION;
	  PositionData1[6].	RelIndexNextPoint	:=  1;
	  PositionData1[6].	MasterPos	:=	        fMasterKeyPos5;
	  PositionData1[6].	SlavePos	:=	       fSaveLength2 ;	
	  PositionData1[6].	SlaveVelo	:=	        (fSaveLength2-fMoveLength)/ (fMasterKeyPos5-fMasterKeyPos4 )	;
*)
	  PositionData1[6].	PointIndex	:=	        6;
	  PositionData1[6].	FunctionType	:=		MOTIONFUNCTYPE_POLYNOM1;
	  PositionData1[6].	PointType	:=	        MOTIONPOINTTYPE_MOTION;
	  PositionData1[6].	RelIndexNextPoint	:=  1;
	  PositionData1[6].	MasterPos	:=	        fMasterKeyPos6;
	  PositionData1[6].	SlavePos	:=	        fSaveLength2;	
	  PositionData1[6].	SlaveVelo	:=	        0	;

	  PositionData1[7].	PointIndex	:=	        7;
	  PositionData1[7].	FunctionType	:=		MOTIONFUNCTYPE_POLYNOM1;
	  PositionData1[7].	PointType	:=	        MOTIONPOINTTYPE_MOTION;
	  PositionData1[7].	RelIndexNextPoint	:=  0;
	  PositionData1[7].	MasterPos	:=	        360;
	  PositionData1[7].	SlavePos	:=	        fSaveLength2;	
	  PositionData1[7].	SlaveVelo	:=	        0	;

     bWriteCamData:=FALSE;
END_IF







(*

IF bWriteCamData  THEN
 
	  Cam_table.ArraySize:=SIZEOF(PositionData1); 
	  Cam_table.NoOfColumns:=1;
	  Cam_table.NoOfRows:=7;
	  Cam_table.pArray:=ADR(PositionData1);
	  Cam_table.TableType:=MC_TABLETYPE_MOTIONFUNCTION;
      //MOTIONFUNCTYPE_BESCHLTRAPEZ     MOTIONFUNCTYPE_POLYNOM7_MM    MOTIONFUNCTYPE_BESCHLTRAPEZ   MOTIONFUNCTYPE_POLYNOM1

	  PositionData1[1].	PointIndex	:=	        1;
	  PositionData1[1].	FunctionType	:=		MOTIONFUNCTYPE_POLYNOM1;//
	  PositionData1[1].	PointType	:=	        MOTIONPOINTTYPE_MOTION;
	  PositionData1[1].	RelIndexNextPoint	:=  1;
	  PositionData1[1].	MasterPos	:=	        0;
	  PositionData1[1].	SlavePos	:=	        0;		//fMoveLength
	  PositionData1[1].	SlaveVelo	:=	        0;
	  
	  PositionData1[2].	PointIndex	:=	        2;
	  PositionData1[2].	FunctionType	:=		MOTIONFUNCTYPE_POLYNOM5_MM;
	  PositionData1[2].	PointType	:=	        MOTIONPOINTTYPE_MOTION;
	  PositionData1[2].	RelIndexNextPoint	:=  1;
	  PositionData1[2].	MasterPos	:=	        fMasterKeyPos1;
	  PositionData1[2].	SlavePos	:=	        0;	
	  PositionData1[2].	SlaveVelo	:=	       0	;

	  PositionData1[3].	PointIndex	:=	        3;
	  PositionData1[3].	FunctionType	:=		MOTIONFUNCTYPE_POLYNOM1;
	  PositionData1[3].	PointType	:=	        MOTIONPOINTTYPE_MOTION;
	  PositionData1[3].	RelIndexNextPoint	:=  0;
	  PositionData1[3].	MasterPos	:=	        fMasterKeyPos2;
	  PositionData1[3].	SlavePos	:=	        fSaveLength1;	
	  PositionData1[3].	SlaveVelo	:=	        0	;

	  PositionData1[4].	PointIndex	:=	        4;
	  PositionData1[4].	FunctionType	:=		MOTIONFUNCTYPE_POLYNOM5_MM;
	  PositionData1[4].	PointType	:=	        MOTIONPOINTTYPE_MOTION;
	  PositionData1[4].	RelIndexNextPoint	:=  1;
	  PositionData1[4].	MasterPos	:=	        fMasterKeyPos3;
	  PositionData1[4].	SlavePos	:=	        fSaveLength1;	
	  PositionData1[4].	SlaveVelo	:=	       0	;

	  PositionData1[5].	PointIndex	:=	        5;
	  PositionData1[5].	FunctionType	:=		MOTIONFUNCTYPE_POLYNOM5_MM;
	  PositionData1[5].	PointType	:=	        MOTIONPOINTTYPE_MOTION;
	  PositionData1[5].	RelIndexNextPoint	:=  1;
	  PositionData1[5].	MasterPos	:=	        fMasterKeyPos4;
	  PositionData1[5].	SlavePos	:=	        fMoveLength;	
	  PositionData1[5].	SlaveVelo	:=	       0	;
(*
	  PositionData1[6].	PointIndex	:=	        6;
	  PositionData1[6].	FunctionType	:=		MOTIONFUNCTYPE_POLYNOM7_MM;
	  PositionData1[6].	PointType	:=	        MOTIONPOINTTYPE_MOTION;
	  PositionData1[6].	RelIndexNextPoint	:=  1;
	  PositionData1[6].	MasterPos	:=	        fMasterKeyPos5;
	  PositionData1[6].	SlavePos	:=	       fSaveLength2 ;	
	  PositionData1[6].	SlaveVelo	:=	        (fSaveLength2-fMoveLength)/ (fMasterKeyPos5-fMasterKeyPos4 )	;
*)
	  PositionData1[6].	PointIndex	:=	        6;
	  PositionData1[6].	FunctionType	:=		MOTIONFUNCTYPE_POLYNOM1;
	  PositionData1[6].	PointType	:=	        MOTIONPOINTTYPE_MOTION;
	  PositionData1[6].	RelIndexNextPoint	:=  1;
	  PositionData1[6].	MasterPos	:=	        fMasterKeyPos6;
	  PositionData1[6].	SlavePos	:=	        0;	
	  PositionData1[6].	SlaveVelo	:=	        0	;

	  PositionData1[7].	PointIndex	:=	        7;
	  PositionData1[7].	FunctionType	:=		MOTIONFUNCTYPE_POLYNOM1;
	  PositionData1[7].	PointType	:=	        MOTIONPOINTTYPE_MOTION;
	  PositionData1[7].	RelIndexNextPoint	:=  0;
	  PositionData1[7].	MasterPos	:=	        360;
	  PositionData1[7].	SlavePos	:=	        0;	
	  PositionData1[7].	SlaveVelo	:=	        0	;

     bWriteCamData:=FALSE;
END_IF

*)
END_ACTION

END_FUNCTION_BLOCK

// ---- P2POUs/BasicFunction/08_Data/CS_Recipe.TcPOU
FUNCTION_BLOCK CS_Recipe
VAR_INPUT
END_VAR
VAR_OUTPUT
END_VAR
VAR
	


 //recipeManCommands: RecipeManCommands;
	result: DWORD;
END_VAR

VAR_IN_OUT
  iRecipe2:    IRecipe;
END_VAR





(*

IF iRecipe2.bCreate THEN
   result:= recipeManCommands.CreateRecipe(RecipeDefinitionName:='Recipes' , RecipeName:='SJ_Rec' );
   iRecipe2.bCreate:=FALSE;
END_IF

IF iRecipe2.bSave THEN
    result:= recipeManCommands.ReadAndSaveRecipeAs(RecipeDefinitionName:='Recipes' , RecipeName:='SJ_Rec' , FileName:='C:\P2Data\P2Par');
    iRecipe2.bSave:=FALSE;
END_IF

IF iRecipe2.bLoad THEN
	result:= RecipeManCommands.LoadFromAndWriteRecipe(RecipeDefinitionName:='Recipes' , RecipeName:='SJ_Rec' , FileName:='C:\P2Data\P2Par');
    iRecipe2.bLoad:=FALSE;
END_IF

*)

END_FUNCTION_BLOCK

// ---- P2POUs/BasicFunction/10_MES/CS_CcdTcp_V2.TcPOU
FUNCTION_BLOCK PUBLIC CS_CcdTcp_V2
VAR_INPUT
END_VAR
VAR_OUTPUT
END_VAR
VAR_IN_OUT
   iCcd2:ICCD;
   Data:STCcdData;
END_VAR


VAR
	ccdDataSend:STCcdDataSend;
	ccdDataReceive:STCcdDataSend;
	fbTcpCon:FB_SocketConnect;
	fbTcpSend:FB_SocketSend;
	fbTcpRec:FB_SocketReceive;
	fbTcpClose: FB_SocketClose;
	bConnect: BOOL;
	bClose: BOOL;
	hTcpSock: T_HSOCKET;
	//aTcpSend:ARRAY[1..10] OF BYTE;
	//aTcpReceive:ARRAY[1..10] OF BYTE;	
	StrSend:STRING;
	StrReceive:STRING;
	fbUdpCreate:FB_SocketUdpCreate;
	hUdp: T_HSOCKET;
	bCreate: BOOL;
	port: UDINT:=9004;
	bSendTcp: BOOL;
	bReceiveTcp: BOOL;
	fbSwingHalt2: MC_Halt;

    strReceiveData: STCcdData;

	iorderTemp: DINT;
	TON100:TON;
END_VAR




	Config();
	
	M_SendReceive();


	
	

	
	
	
	

	
	
	
	
	
	
	
	
	
	
	
	
	
	
	
	
	
(*	
   fbUdpCreate(
	sSrvNetId:= , 
	sLocalHost:= , 
	nLocalPort:= port, 
	bExecute:=bCreate , 
	tTimeout:= , 
	bBusy=> , 
	bError=> , 
	nErrId=> , 
	hSocket=> hUdp);
	
	
	*)

ACTION Config:



  IF iCcd2.bComOpen THEN
	 bConnect:=TRUE;	
	 bClose:=FALSE;
	 iCcd2.bComOpen:=FALSE;
  END_IF
  
   IF iCcd2.bComClose THEN
	 bConnect:=FALSE;	
	 bClose:=TRUE;
	 iCcd2.bComClose:=FALSE;
  END_IF 
  
  
  
fbTcpCon(
	sSrvNetId:= ''   ,          //       (*'169.254.46.193.1.1'*) , 
	sRemoteHost:='192.168.2.11'     , 
	nRemotePort:= 2020, 
	bExecute:=bConnect , 
	tTimeout:= , 
	bBusy=> , 
	bError=> , 
	nErrId=> , 
	hSocket=>hTcpSock );
	
fbTcpClose(
	sSrvNetId:= ''   , 
	hSocket:=hTcpSock , 
	bExecute:=bClose , 
	tTimeout:=T#5S , 
	bBusy=> , 
	bError=> , 
	nErrId=> );


IF fbTcpCon.bBusy THEN
	bConnect:=FALSE;
END_IF

IF fbTcpClose.bBusy THEN
   bClose:=FALSE;
END_IF
END_ACTION

ACTION M_SendReceive:



  IF iCcd2.bSend THEN
	 bSendTcp:=TRUE;
	 iCcd2.bDone:=FALSE;
	 iCcd2.bError:=FALSE;
	 //iCcd2.strReceive:='';
    MEMSET(ADR(ccdDataSend.strBetryName),0,SIZEOF(ccdDataSend.strBetryName));
	MEMSET(ADR(ccdDataSend.strCode),0,SIZEOF(ccdDataSend.strCode));
	MEMSET(ADR(ccdDataSend.strShortData),0,SIZEOF(ccdDataSend.strShortData));
	MEMSET(ADR(ccdDataSend.strHotPress),0,SIZEOF(ccdDataSend.strHotPress));
    STRING_TO_UTF8(pDstUTF8:=ADR(ccdDataSend.strBetryName) , pSrcSTRING:=ADR(Data.strBetryName) , nDstSize:=INT_TO_UINT( LEN(STR:=Data.strBetryName )+1) );
    STRING_TO_UTF8(pDstUTF8:=ADR(ccdDataSend.strCode) , pSrcSTRING:=ADR(Data.strCode) , nDstSize:=INT_TO_UINT( LEN(STR:=Data.strCode )+1) ); 
    STRING_TO_UTF8(pDstUTF8:=ADR(ccdDataSend.strShortData) , pSrcSTRING:=ADR(Data.strShortData) , nDstSize:=INT_TO_UINT( LEN(STR:=Data.strShortData )+1) );
	STRING_TO_UTF8(pDstUTF8:=ADR(ccdDataSend.strHotPress) , pSrcSTRING:=ADR(Data.strHotPress) , nDstSize:=INT_TO_UINT( LEN(STR:=Data.strHotPress )+1) );
    iCcd2.bSend:=FALSE;
	iorderTemp:=Data.iorder;
	TON100.IN:=TRUE;
END_IF
	 
fbTcpSend(
		sSrvNetId:= , 
		hSocket:=hTcpSock , 
		cbLen:=SIZEOF(ccdDataSend), 
		pSrc:= ADR(ccdDataSend), 
		bExecute:= bSendTcp, 
		tTimeout:= T#2S , 
		bBusy=> , 
		bError=> , 
		nErrId=> );
	IF bSendTcp AND fbTcpSend.bBusy THEN
		bSendTcp:=FALSE;
	END_IF
	
	
bReceiveTcp:=NOT bReceiveTcp;
	
fbTcpRec(
	sSrvNetId:= , 
	hSocket:= hTcpSock, 
	cbLen:=SIZEOF(ccdDataReceive) , 
	pDest:=ADR(ccdDataReceive) , 
	bExecute:=bReceiveTcp , 
	tTimeout:= T#5S, 
	bBusy=> , 
	bError=> , 
	nErrId=> , 
	nRecBytes=> );

	
TON100(IN:= , PT:= T#3S, Q=> , ET=> );//通讯超时
	
 ccdDataReceive.iorder;	//功能码 2     3      4
 UTF8_TO_STRING (pDstSTRING:= ADR(strReceiveData.strBetryName) , pSrcUTF8:= ADR(ccdDataReceive.strBetryName), nDstSize:=SIZEOF(ccdDataReceive.strBetryName) , nDstLen=> );//文件名

	IF ccdDataReceive.iorder=iorderTemp  AND ccdDataReceive.iorder>0  THEN  //发送对应 返回功能码  
		
        IF ccdDataReceive.iorder=2 THEN     //给MES发送数据成功
		    iCcd2.bDone:=TRUE; 
		ELSIF ccdDataReceive.iorder=3 THEN   //取料请求文件名成功  有可能文件名是空
			IF strReceiveData.strBetryName='' THEN //文件名空  给plc自定义文件名   也可以做报警    
			   iCcd2.bDone:=TRUE; 
			    iCcd2.strReceive:= MAIN.strTime;
			ELSE
			 iCcd2.strReceive:= strReceiveData.strBetryName;
			  iCcd2.bDone:=TRUE; 
			END_IF
		ELSIF ccdDataReceive.iorder=4 THEN   //取料夹爪夹空   不用处理文件名字
		    iCcd2.bDone:=TRUE; 
			iCcd2.strReceive:='';
		END_IF
	
	   MEMSET(ADR(ccdDataReceive),0,SIZEOF(ccdDataReceive));
	   iorderTemp:=0;
	   TON100.IN:=FALSE;
	END_IF
	
	IF TON100.Q AND iorderTemp<>0 THEN  //通讯超时报警
		   ;           //报警信号
		 TON100.IN:=FALSE;
		  iorderTemp:=0;
	END_IF
END_ACTION

END_FUNCTION_BLOCK

// ---- P3POUs/P3FB/ADSWrite_Limit.TcPOU
FUNCTION_BLOCK ADSWrite_Limit
VAR_INPUT
	IDXGRP_W:UDINT;//ADS组别索引
	IDXOFFS_W:UDINT;//ADS补偿索引
	IDXOFFSLimit_W:UDINT;//ADS软限位开关补偿索引
	bSetButton:BOOL;(*ADS软限位值写入*)
	bSetLimitButton:BOOL;(*ADS软限位开关*)
	fSavePositionBias:LREAL;
	AxisNo:UINT;
	ADSMark:BOOL;//
END_VAR
VAR_IN_OUT
	
END_VAR
VAR_OUTPUT
	bWriteAlarm:BOOL;//
	fSaveBias:LREAL;
END_VAR
VAR
	Step_W_Date :UINT;
	fbADSwrite: ADSWRITE;(*ADS写功能块定义*)
	fbADSRead: ADSRead;//ADS写入功能块
	rADSWrite: R_TRIG;(*ADS写完成上升沿*)
	rADSRead: R_TRIG;(*ADS写完成上升沿*)
	rSetButton:R_TRIG;(*ADS写变量的上升沿*)
	R_SetLimitButton: R_TRIG;//软限位开关出发上升沿
	F_SetLimitButton: F_TRIG;//软限位开关出发下降沿
	R_ADSMark:R_TRIG;
	bFirstCycle:BOOL;//首次上电
	WriteNGcount:INT;
END_VAR

R_ADSMark(CLK:=ADSMark , Q=> );
IF R_ADSMark.Q THEN
	bFirstCycle:=TRUE;//首次上电
END_IF
CASE Step_W_Date OF
0:
	rSetButton(CLK:=bSetButton , Q=> );
	R_SetLimitButton(CLK:=bSetLimitButton , Q=> );
	F_SetLimitButton(CLK:=bSetLimitButton , Q=> );
	WriteNGcount:=0;
	IF rSetButton.Q OR bFirstCycle THEN
		bSetButton:=FALSE;
		bWriteAlarm:=FALSE;//
		Step_W_Date:=50;
	ELSIF R_SetLimitButton.Q OR F_SetLimitButton.Q THEN
			bWriteAlarm:=FALSE;//
		Step_W_Date:=450;
	END_IF
50:
	//arrAxisCtrl[AxisNo].Cmd.bEnable:=FALSE;
	Step_W_Date:=100;
100:
	fbADSwrite.LEN:=8;
	fbADSwrite.SRCADDR:=ADR(fSavePositionBias);
	fbADSwrite.IDXOFFS:=IDXOFFS_W;
	Step_W_Date:=150;
150:
	fbADSwrite.WRITE:=TRUE;
	rADSWrite(CLK:=NOT fbADSwrite.BUSY , Q=> );
	IF rADSWrite.Q THEN
		fbADSwrite.WRITE:=FALSE;
		Step_W_Date:=200;
	ELSIF fbADSwrite.ERR THEN
		bWriteAlarm:=TRUE;
		Step_W_Date:=0;
	END_IF
	
200:
	fbADSRead.LEN:=8;
	fbADSRead.DESTADDR:=ADR(fSaveBias);
	fbADSRead.IDXOFFS:=IDXOFFS_W;
	Step_W_Date:=250;
	
250:
	fbADSRead.READ:=TRUE;
	rADSRead(CLK:=NOT fbADSRead.BUSY , Q=> );
	IF rADSRead.Q THEN
		fbADSRead.READ:=FALSE;
		Step_W_Date:=300;
	END_IF
	
300:
	IF fSaveBias=fSavePositionBias THEN
		Step_W_Date:=400;
	ELSE
		WriteNGcount:=WriteNGcount+1;
		Step_W_Date:=350;	
	END_IF
350:
	IF  WriteNGcount<=1 THEN
		Step_W_Date:=50;
	ELSE
		Step_W_Date:=400;
	END_IF
400:
	IF bFirstCycle THEN
		Step_W_Date:=450;
	ELSE
		Step_W_Date:=0;
	END_IF
	
	
450://软限位开关
	bFirstCycle:=FALSE;//首次上电
	//arrAxisCtrl[AxisNo].Cmd.bEnable:=FALSE;
	Step_W_Date:=500;
500:
	fbADSwrite.LEN:=2;
	fbADSwrite.SRCADDR:=ADR(bSetLimitButton);
	fbADSwrite.IDXOFFS:=IDXOFFSLimit_W;
	Step_W_Date:=550;
550:
	fbADSwrite.WRITE:=TRUE;
	rADSWrite(CLK:=NOT fbADSwrite.BUSY , Q=> );
	IF rADSWrite.Q THEN
		fbADSwrite.WRITE:=FALSE;
		Step_W_Date:=600;
	ELSIF fbADSwrite.ERR THEN
		bWriteAlarm:=TRUE;
		Step_W_Date:=0;
	END_IF

600:
	IF NOT  bFirstCycle THEN
 		Step_W_Date:=0;
	END_IF
	
END_CASE
 	





fbADSwrite(
	NETID:='' , 
	PORT:=501 , 
	IDXGRP:=IDXGRP_W, 
	IDXOFFS:=, 
	LEN:= , 
	SRCADDR:=, 
	WRITE:= , 
	TMOUT:=T#500MS , 
	BUSY=> , 
	ERR=> , 
	ERRID=>
);
 
fbADSRead(
	NETID:= , 
	PORT:=501 , 
	IDXGRP:= IDXGRP_W, 
	IDXOFFS:= , 
	LEN:= , 
	DESTADDR:= , 
	READ:= , 
	TMOUT:=T#500MS , 
	BUSY=> , 
	ERR=> , 
	ERRID=> );

END_FUNCTION_BLOCK

// ---- P3POUs/P3FB/FB_HDData.TcPOU
FUNCTION_BLOCK FB_HDData
VAR_INPUT
	
    Alm :    BOOL ;//报警
	Wait :BOOL ;//待机
	Run :BOOL ;//运行
	XL_Wait:BOOL ;//下料等待时间
	Query:BOOL;//时间查询
	

END_VAR
VAR_OUTPUT
		STTimedata:ARRAY[0..32] OF ST_Timedata_1;

END_VAR
VAR
	
	rRun : R_TRIG;
	rAlm : R_TRIG;
	rWait : R_TRIG;
	rXL_Wait : R_TRIG;
	
	fRun: F_TRIG;
	fAlm: F_TRIG;
	fWait: F_TRIG;
    delay:BOOL ;//延时
	TON_1: TON;
	i:INT;
	K: INT;
	J: BOOL;
END_VAR

VAR_IN_OUT
     date1:INT;//查询日期
END_VAR

K:=K+1;
	IF K>499THEN
		J:=TRUE;
		K:=0;
	ELSE
		J:=FALSE;
	END_IF




///////////////运行时间/////////////////
rRun(CLK:= J , Q=> );

IF rRun.Q  AND  Run THEN
	STTimedata[system.stTime.wDay].RunTime[system.stTime.wHour]:=STTimedata[system.stTime.wDay].RunTime[system.stTime.wHour]+1;
END_IF

IF STTimedata[system.stTime.wDay].RunTime[system.stTime.wHour]> 3600 THEN
	STTimedata[system.stTime.wDay].RunTime[system.stTime.wHour]:= 3600 ;
END_IF

//IF STTimedata[system.stTime.wDay].AlmTime[system.stTime.wHour]= 0 AND STTimedata[system.stTime.wDay].WaitTime[system.stTime.wHour]= 0  AND 
   // (STTimedata[system.stTime.wDay].RunTime[system.stTime.wHour]= 3585  OR  STTimedata[system.stTime.wDay].RunTime[system.stTime.wHour]= 3586 ) THEN
	//STTimedata[system.stTime.wDay].RunTime[system.stTime.wHour]:= 3600 ;
//END_IF


///////////////待机时间///////////////
rWait(CLK:=J , Q=> );

IF rWait.Q  AND Wait THEN
	STTimedata[system.stTime.wDay].WaitTime[system.stTime.wHour]:=STTimedata[system.stTime.wDay].WaitTime[system.stTime.wHour]+1;
END_IF

IF STTimedata[system.stTime.wDay].WaitTime[system.stTime.wHour]> 3600 THEN
	STTimedata[system.stTime.wDay].WaitTime[system.stTime.wHour]:= 3600 ;
END_IF

//IF STTimedata[system.stTime.wDay].RunTime[system.stTime.wHour]= 0 AND STTimedata[system.stTime.wDay].AlmTime[system.stTime.wHour]= 0  AND 
  //   (STTimedata[system.stTime.wDay].RunTime[system.stTime.wHour]= 3585  OR  STTimedata[system.stTime.wDay].RunTime[system.stTime.wHour]= 3586 )  THEN
//	STTimedata[system.stTime.wDay].WaitTime[system.stTime.wHour]:= 3600 ;
//END_IF


////////////////报警时间///////////////
rAlm(CLK:=J , Q=> );

IF rAlm.Q AND Alm THEN
	STTimedata[system.stTime.wDay].AlmTime[system.stTime.wHour]:=STTimedata[system.stTime.wDay].AlmTime[system.stTime.wHour]+1;
END_IF

IF STTimedata[system.stTime.wDay].AlmTime[system.stTime.wHour]> 3600 THEN
	STTimedata[system.stTime.wDay].AlmTime[system.stTime.wHour]:= 3600 ;
END_IF

//IF STTimedata[system.stTime.wDay].RunTime[system.stTime.wHour]= 0 AND STTimedata[system.stTime.wDay].WaitTime[system.stTime.wHour]= 0  AND
 ////   (STTimedata[system.stTime.wDay].RunTime[system.stTime.wHour]= 3585  OR  STTimedata[system.stTime.wDay].RunTime[system.stTime.wHour]= 3586 ) THEN
//	STTimedata[system.stTime.wDay].AlmTime[system.stTime.wHour]:= 3600 ;
//END_IF

////////////////下料等待托盘时间///////////////
rXL_Wait(CLK:=J, Q=> );

IF rXL_Wait.Q AND XL_Wait THEN
	STTimedata[system.stTime.wDay].XLWaitTime[system.stTime.wHour]:=STTimedata[system.stTime.wDay].XLWaitTime[system.stTime.wHour]+1;
END_IF

//数据查询
IF Query THEN
	delay:=TRUE;
END_IF

TON_1(IN:= , PT:=T#60S , Q=> , ET=> );
IF delay THEN
		  IF NOT TON_1.Q THEN
			  TON_1.IN:=TRUE;
		  ELSE	
			  delay:=FALSE;
			  date1:=system.stTime.wDay;
		  END_IF	 
ELSE	
	 TON_1.IN:=FALSE;
END_IF


IF NOT delay THEN
STTimedata[32]:=STTimedata[system.stTime.wDay];
ELSE
STTimedata[32]:=STTimedata[date1];
END_IF

//数据清零
IF (system.stTime.wMonth=2 AND  system.stTime.wDay=28 )   OR
    ((system.stTime.wMonth=4 OR system.stTime.wMonth=6 OR system.stTime.wMonth=9 OR system.stTime.wMonth=11) AND system.stTime.wDay=30 )   OR
	((system.stTime.wMonth=1 OR  system.stTime.wMonth=3 OR system.stTime.wMonth=5 OR system.stTime.wMonth=7 OR system.stTime.wMonth=8 OR system.stTime.wMonth=10 OR system.stTime.wMonth=12) AND  system.stTime.wDay=31)  AND
    system.stTime.wHour=23 AND  system.stTime.wMinute=59 AND system.stTime.wSecond =59 THEN
	FOR i:=0 TO 32  DO
	MEMSET(ADR(STTimedata[i]),0,SIZEOF(STTimedata[i]));	
	END_FOR
END_IF

END_FUNCTION_BLOCK

// ---- P3POUs/P3FB/FB_OEE.TcPOU
FUNCTION_BLOCK FB_OEE
VAR_INPUT
	
    Alm :    BOOL ;//报警
	Wait :BOOL ;//待机
	Run :BOOL ;//运行

	

END_VAR
VAR_OUTPUT
		OEE:REAL;//稼动率
       
END_VAR
VAR
	 STTimedata:ST_Timedata_1;
	rRun : R_TRIG;
	rAlm : R_TRIG;
	rWait : R_TRIG;
	rXL_Wait : R_TRIG;
	
	fRun: F_TRIG;
	fAlm: F_TRIG;
	fWait: F_TRIG;
    delay:BOOL ;//延时
	TON_1: TON;
	i:INT;
	K: INT;
	J: BOOL;
	MalfunctionTime:REAL;//报警时间
	RunTime1:REAL;//运行时间

END_VAR

VAR_IN_OUT
   
END_VAR

K:=K+1;
	IF K>499THEN
		J:=TRUE;
		K:=0;
	ELSE
		J:=FALSE;
	END_IF




///////////////运行时间/////////////////
rRun(CLK:= J , Q=> );

IF rRun.Q  AND  Run THEN
	STTimedata.RunTime[HMI_Hour]:=STTimedata.RunTime[HMI_Hour]+1;
END_IF

IF STTimedata.RunTime[HMI_Hour]> 3600 THEN
	STTimedata.RunTime[HMI_Hour]:= 3600 ;
END_IF




///////////////待机时间///////////////
rWait(CLK:=J , Q=> );

IF rWait.Q  AND Wait THEN
	STTimedata.WaitTime[HMI_Hour]:=STTimedata.WaitTime[HMI_Hour]+1;
END_IF

IF STTimedata.WaitTime[HMI_Hour]> 3600 THEN
	STTimedata.WaitTime[HMI_Hour]:= 3600 ;
END_IF

IF STTimedata.RunTime[HMI_Hour]= 0 AND STTimedata.AlmTime[HMI_Hour]= 0  AND 
     (STTimedata.RunTime[HMI_Hour]= 3585  OR  STTimedata.RunTime[HMI_Hour]= 3586 )  THEN
//	STTimedata[HMI_day].WaitTime[HMI_Hour]:= 3600 ;
END_IF


////////////////报警时间///////////////
rAlm(CLK:=J , Q=> );

IF rAlm.Q AND Alm THEN
	STTimedata.AlmTime[HMI_Hour]:=STTimedata.AlmTime[HMI_Hour]+1;
END_IF

IF STTimedata.AlmTime[HMI_Hour]> 3600 THEN
	STTimedata.AlmTime[HMI_Hour]:= 3600 ;
END_IF

IF STTimedata.RunTime[HMI_Hour]= 0 AND STTimedata.WaitTime[HMI_Hour]= 0  AND
    (STTimedata.RunTime[HMI_Hour]= 3585  OR  STTimedata.RunTime[HMI_Hour]= 3586 ) THEN
//	STTimedata[HMI_day].AlmTime[HMI_Hour]:= 3600 ;
END_IF

IF   HMI_Hour=23 AND  HMI_Minute=59 AND  HMI_Second=59 THEN
	FOR i:=0 TO 23  DO
   STTimedata.RunTime[i]:=0	;
   STTimedata.AlmTime[i]:=0	;
   STTimedata.WaitTime[i]:=0;
	END_FOR
END_IF

//稼动率
RunTime1:=STTimedata.RunTime[0]+STTimedata.RunTime[1]+STTimedata.RunTime[2]+STTimedata.RunTime[3]+STTimedata.RunTime[4]+
                      STTimedata.RunTime[5]+STTimedata.RunTime[6]+STTimedata.RunTime[7]+STTimedata.RunTime[8]+STTimedata.RunTime[9]+
                      STTimedata.RunTime[10]+STTimedata.RunTime[11]+STTimedata.RunTime[12]+STTimedata.RunTime[13]+STTimedata.RunTime[14]+
                      STTimedata.RunTime[15]+STTimedata.RunTime[16]+STTimedata.RunTime[17]+STTimedata.RunTime[18]+STTimedata.RunTime[19]+
					  STTimedata.RunTime[20]+STTimedata.RunTime[21]+STTimedata.RunTime[22]+STTimedata.RunTime[23];
					  
MalfunctionTime:=STTimedata.AlmTime[0]+STTimedata.AlmTime[1]+STTimedata.AlmTime[2]+STTimedata.AlmTime[3]+	STTimedata.AlmTime[4]+				  
					              STTimedata.AlmTime[5]+STTimedata.AlmTime[6]+STTimedata.AlmTime[7]+STTimedata.AlmTime[8]+	STTimedata.AlmTime[9]+		
					              STTimedata.AlmTime[10]+STTimedata.AlmTime[11]+STTimedata.AlmTime[12]+STTimedata.AlmTime[13]+	STTimedata.AlmTime[14]+		
					              STTimedata.AlmTime[15]+STTimedata.AlmTime[16]+STTimedata.AlmTime[17]+STTimedata.AlmTime[18]+	STTimedata.AlmTime[19]+		
								  STTimedata.AlmTime[20]+STTimedata.AlmTime[21]+STTimedata.AlmTime[22]+STTimedata.AlmTime[23];
IF RunTime1>0 THEN								  
OEE:=	(RunTime1/(RunTime1+	MalfunctionTime	))*100	;			 
END_IF

END_FUNCTION_BLOCK

// ---- P2POUs/BasicFunction/01_IO/ScaleTrans_1.TcPOU
FUNCTION ScaleTrans_1 : REAL
VAR_INPUT
	EN:BOOL;//启动条件
	Scalln:REAL;//输入值
	X0:REAL;//输入范围下限值
	Y0:REAL;//输出范围下限值
	X1:REAL;//输入范围上限值
	Y1:REAL;//输出范围上限值
	Sclofs:REAL;//偏置值
END_VAR
VAR
END_VAR

IF EN THEN
	IF (X1-X0)<> 0 THEN
		ScaleTrans:=(Y1-Y0)/(X1-X0)*(Scalln-X0)+Y0+Sclofs;
	END_IF
END_IF

END_FUNCTION

// ---- P2POUs/BasicFunction/02_SystemCheck/CheckBounds.TcPOU
// 隐含生成代码：不要编辑
FUNCTION CheckBounds : DINT
VAR_INPUT
	index, lower, upper: DINT;
END_VAR

// 隐含生成代码：这里只是对代码实现的建议
{noflow}
IF  index < lower THEN
	CheckBounds := lower;
ELSIF  index > upper THEN
	CheckBounds := upper;
ELSE  
	CheckBounds := index;
END_IF
{flow}

END_FUNCTION

// ---- P2POUs/BasicFunction/02_SystemCheck/CheckDivDInt.TcPOU
// 隐含生成代码：不要编辑
FUNCTION CheckDivDInt : DINT
VAR_INPUT
	divisor:DINT;
END_VAR

// 隐含生成代码：这里只是对代码实现的建议
{noflow}
IF divisor = 0 THEN
	CheckDivDInt:=1;
ELSE
	CheckDivDInt:=divisor;
END_IF;
{flow}

END_FUNCTION

// ---- P2POUs/BasicFunction/02_SystemCheck/CheckDivLInt.TcPOU
// 隐含生成代码：不要编辑
FUNCTION CheckDivLInt : LINT
VAR_INPUT
	divisor:LINT;
END_VAR

// 隐含生成代码：这里只是对代码实现的建议
{noflow}
IF divisor = 0 THEN
	CheckDivLInt:=1;
ELSE
	CheckDivLInt:=divisor;
END_IF;
{flow}

END_FUNCTION

// ---- P2POUs/BasicFunction/02_SystemCheck/CheckDivLReal.TcPOU
// 隐含生成代码：不要编辑
FUNCTION CheckDivLReal : LREAL
VAR_INPUT
	divisor:LREAL;
END_VAR

// 隐含生成代码：这里只是对代码实现的建议
{noflow}
IF divisor = 0 THEN
	CheckDivLReal:=1;
ELSE
	CheckDivLReal:=divisor;
END_IF;
{flow}

END_FUNCTION

// ---- P2POUs/BasicFunction/02_SystemCheck/CheckDivReal.TcPOU
// 隐含生成代码：不要编辑
FUNCTION CheckDivReal : REAL
VAR_INPUT
	divisor:REAL;
END_VAR

// 隐含生成代码：这里只是对代码实现的建议
{noflow}
IF divisor = 0 THEN
	CheckDivReal:=1;
ELSE
	CheckDivReal:=divisor;
END_IF;
{flow}

END_FUNCTION

// ---- P2POUs/BasicFunction/02_SystemCheck/CheckLRangeSigned.TcPOU
// 隐含生成代码：不要编辑
FUNCTION CheckLRangeSigned : LINT
VAR_INPUT
	value, lower, upper: LINT;
END_VAR

// 隐含生成代码：这里只是对代码实现的建议
{noflow}
IF (value < lower) THEN
	CheckLRangeSigned := lower;
ELSIF(value > upper) THEN
	CheckLRangeSigned := upper;
ELSE
	CheckLRangeSigned := value;
END_IF

{flow}

END_FUNCTION

// ---- P2POUs/BasicFunction/02_SystemCheck/CheckLRangeUnsigned.TcPOU
// 隐含生成代码：不要编辑
FUNCTION CheckLRangeUnsigned : ULINT
VAR_INPUT
	value, lower, upper: ULINT;
END_VAR

// 隐含生成代码：这里只是对代码实现的建议
{noflow}
IF (value < lower) THEN
	CheckLRangeUnsigned := lower;
ELSIF(value > upper) THEN
	CheckLRangeUnsigned := upper;
ELSE
	CheckLRangeUnsigned := value;
END_IF
{flow}

END_FUNCTION

// ---- P2POUs/BasicFunction/02_SystemCheck/CheckPointer.TcPOU
// 隐含生成代码：不要编辑
FUNCTION CheckPointer : POINTER TO BYTE
VAR_INPUT 
	ptToTest : POINTER TO BYTE; // 指针的目标地址
	iSize : DINT;		        // 指针指向的类型大小。（例如：POINTER TO ARRAY [0..9] OF INT为20）
	iGran : DINT;		        // 指针访问的粒度，即指针指向的类型中最大的非结构数据类型的大小。（例如：POINTER TO ARRAY [0..9] OF INT为2）
	bWrite: BOOL;		        // 指示读或写权限。TRUE=写权限。
END_VAR

// 隐含生成代码：这里只是对代码实现的建议
{noflow}
IF ptToTest=0 THEN
    ADSLOGSTR(ADSLOG_MSGTYPE_ERROR OR ADSLOG_MSGTYPE_STRING,'CheckPointer failed due to invalid address.','');
ELSIF iSize<=0 THEN
    ADSLOGSTR(ADSLOG_MSGTYPE_ERROR OR ADSLOG_MSGTYPE_STRING,'CheckPointer failed due to invalid size.','');
ELSIF iGran<=0 THEN
    ADSLOGSTR(ADSLOG_MSGTYPE_ERROR OR ADSLOG_MSGTYPE_STRING,'CheckPointer failed due to invalid granularity.','');
// -> Please note that the following memory area check is time consuming:
//ELSIF F_CheckMemoryArea(pData:=ptToTest,nSize:=DINT_TO_UDINT(iSize)) = E_TcMemoryArea.Unknown THEN
//    ADSLOGSTR(ADSLOG_MSGTYPE_ERROR OR ADSLOG_MSGTYPE_STRING,'CheckPointer failed due to unknown memory area.','');
END_IF
CheckPointer := ptToTest;
{flow}

END_FUNCTION

// ---- P2POUs/BasicFunction/02_SystemCheck/CheckRangeSigned.TcPOU
// 隐含生成代码：不要编辑
FUNCTION CheckRangeSigned : DINT
VAR_INPUT
	value, lower, upper: DINT;
END_VAR

// 隐含生成代码：这里只是对代码实现的建议
{noflow}
IF (value < lower) THEN
	CheckRangeSigned := lower;
ELSIF(value > upper) THEN
	CheckRangeSigned := upper;
ELSE
	CheckRangeSigned := value;
END_IF
{flow}

END_FUNCTION

// ---- P2POUs/BasicFunction/02_SystemCheck/CheckRangeUnsigned.TcPOU
// 隐含生成代码：不要编辑
FUNCTION CheckRangeUnsigned : UDINT
VAR_INPUT
	value, lower, upper: UDINT;
END_VAR

// 隐含生成代码：这里只是对代码实现的建议
{noflow}
IF (value < lower) THEN
	CheckRangeUnsigned := lower;
ELSIF(value > upper) THEN
	CheckRangeUnsigned := upper;
ELSE
	CheckRangeUnsigned := value;
END_IF
{flow}

END_FUNCTION

// ---- P2POUs/BasicFunction/03_Motion/Three_Scale.TcPOU
FUNCTION Three_Scale : REAL
VAR_INPUT
	X:REAL;
	Sall: REAL;
	T:REAL;
END_VAR
VAR
	a2: REAL;
	a3: REAL;
END_VAR

a2:=3*Sall/EXPT(T,REAL#2);
a3:=-2*Sall/EXPT(T,REAL#3);
Three_Scale:=a3*EXPT(X,REAL#3) + a2*EXPT(X,REAL#2);

END_FUNCTION

// ---- P2POUs/BasicFunction/05_Actuators/FB_CylinderV2.TcPOU
FUNCTION_BLOCK FB_CylinderV2
VAR_INPUT
	bReset	:	BOOL	;	
END_VAR

VAR_IN_OUT
  CyCtrl: ST_CyCtrl;
END_VAR


VAR
	rON	:	R_TRIG	;
	rOFF	:	R_TRIG	;
	rFree	:	R_TRIG	;
	Delay2	:	TON	;
	Delay3	:	TON	;
	RS1	:	RS	;
	RS2	:	RS	;
	Delay4	:	TON	;
	Delay5	:	TON	;
	rError1	:	R_TRIG	;
	fError2	:	F_TRIG	;
	fError1	:	F_TRIG	;
	rError2	:	R_TRIG	;
	DelayOnSwitch	:	TON	;
	DelayOffSwitch	:	TON	;
	M1	:	BOOL	;



END_VAR


rON(CLK:=CyCtrl.Cmd.bON );   
rOFF(CLK:=CyCtrl.Cmd.bOFF  );
rFree(CLK:=CyCtrl.Cmd.bFree  );

IF rON.Q THEN 
	CyCtrl.Cmd.bOFF:=FALSE;
    CyCtrl.Cmd.bFree :=FALSE;
END_IF;
IF rOFF.Q THEN 
	CyCtrl.Cmd.bON:=FALSE;
    CyCtrl.Cmd.bFree :=FALSE;
END_IF;
IF rFree.Q THEN 
	CyCtrl.Cmd.bON:=FALSE;
	CyCtrl.Cmd.bOFF:=FALSE;
END_IF;
;

IF   CyCtrl.Cmd.iType=1 OR CyCtrl.Cmd.iType=3   THEN  // 双
		IF   rON.Q THEN
				RS1.SET:=TRUE;
		        RS1.RESET1:=FALSE;
				RS2.SET:=FALSE;
		        RS2.RESET1:=TRUE;			
		END_IF;
		IF   rOFF.Q THEN
				RS2.SET:=TRUE;
		        RS2.RESET1:=FALSE;
				RS1.SET:=FALSE;
		       RS1.RESET1:=TRUE;		   
		END_IF;
END_IF;	

IF   CyCtrl.Cmd.iType=2  OR  CyCtrl.Cmd.iType=4   THEN  //   单
		IF   rON.Q THEN
				RS1.SET:=TRUE;
		       RS1.RESET1:=FALSE;
		END_IF;
		IF   rOFF.Q THEN
				RS1.SET:=FALSE;
		       RS1.RESET1:=TRUE;
		END_IF;
   
   	 RS2.SET:=FALSE;
	 RS2.RESET1:=TRUE;	  
END_IF;
  
IF  CyCtrl.Cmd.iType>=1 AND   CyCtrl.Cmd.iType<=3 THEN  //泄压
 	 IF   rFree.Q THEN
		RS1.SET:=FALSE;
		RS1.RESET1:=TRUE;		
		RS2.SET:=FALSE;
		RS2.RESET1:=TRUE;
   END_IF
END_IF

IF  CyCtrl.Cmd.iType=1 OR  CyCtrl.Cmd.iType=2 THEN
     CyCtrl.Status.ONState:=CyCtrl.Io.DIOnSwitch;
      CyCtrl.Status.OFFState:=CyCtrl.Io.DIOFFSwitch;
END_IF
IF  CyCtrl.Cmd.iType=4  THEN  
     CyCtrl.Status.ONState:=  CyCtrl.Io.DOStatus1;
      CyCtrl.Status.OFFState:=NOT CyCtrl.Io.DOStatus1;
END_IF
IF  CyCtrl.Cmd.iType=3  THEN  
     CyCtrl.Status.ONState:=CyCtrl.Io.DOStatus1;
      CyCtrl.Status.OFFState:=CyCtrl.Io.DOStatus2;
END_IF


//仿真用
//DelayOnSwitch(IN:=CyCtrl.Io.DOStatus1 , PT:=T#2000MS  );  //仿真用
//DelayOffSwitch(IN:=CyCtrl.Io.DOStatus2 , PT:=T#2000MS  );

//CyCtrl.Status.ONState:=DelayOnSwitch.Q;
//CyCtrl.Status.OFFState:=DelayOffSwitch.Q;
   
RS1( Q1=>CyCtrl.Io.DOStatus1 );
RS2( Q1=>CyCtrl.Io.DOStatus2 );
///////////////////////////////////////
IF  CyCtrl.Cmd.iType=2 OR  CyCtrl.Cmd.iType=4  THEN  //   单控 T#100MS
	Delay4(IN:=(RS1.SET      AND  NOT  CyCtrl.Status.ONState) , PT:=INT_TO_TIME(CyCtrl.Cmd.ErrorTime)*1000  );//ON 到位报警
	Delay5(IN:=(RS1.RESET1 AND NOT  CyCtrl.Status.OFFState ) , PT:= INT_TO_TIME(CyCtrl.Cmd.ErrorTime)*1000  );//OFF 到位报警
	;
ELSIF  CyCtrl.Cmd.iType=1  OR  CyCtrl.Cmd.iType=3  THEN
	Delay4(IN:=(RS1.SET      AND  NOT  CyCtrl.Status.ONState) ,   PT:= INT_TO_TIME(CyCtrl.Cmd.ErrorTime)*1000     );//ON 到位报警
	Delay5(IN:=(RS2.SET      AND  NOT  CyCtrl.Status.OFFState ) , PT:=INT_TO_TIME(CyCtrl.Cmd.ErrorTime)*1000      );//OFF 到位报警 MULTIME(In1:=T#100MS, In2:=ErrorTime) 
	;
END_IF;
	
CyCtrl.Status.Error1:=Delay4.Q;
CyCtrl.Status.Error2:=Delay5.Q;




(*

rError1(CLK:=Delay4.Q  );  
rError2(CLK:=Delay5.Q  );  

IF rError1.Q THEN    
	CyCtrl.Status.Error1:=TRUE;
END_IF;

IF rError2.Q THEN    
	CyCtrl.Status.Error2:=TRUE;
END_IF;


IF bReset AND (  CyCtrl.Status.Error1 OR CyCtrl.Status.Error2 )THEN
	CyCtrl.Status.Error1:=FALSE;
	CyCtrl.Status.Error2:=FALSE;
END_IF;

*)

END_FUNCTION_BLOCK

// ---- P2POUs/BasicFunction/08_Data/CS_Data_Test.TcPOU
FUNCTION_BLOCK CS_Data_Test
VAR_INPUT
END_VAR
VAR_OUTPUT
END_VAR
VAR
	//tDataSave:TON;
	//fbSaveData:FB_WritePersistentData;
	//fbXMLWrite:FB_XMLSrvWrite;
	//bWriteXml: BOOL;
	
	fbFileOpen_w:fb_fileopen;
	//fbFileOpen_r:fb_fileopen;
	fbFileWrite:fb_filewrite;
	fbFileRead:FB_FileRead;
	fbFileClose_w:fb_FileClose;
	//fbFileClose_r:fb_FileClose;
	HFILE:UINT;
	//HFILE_R:UINT;
	//bFileOpen_w:BOOL;
	//bFileOpen_r:BOOL;
	//bFileWrite:BOOL;
	//bFileClose_w:BOOL;
	//bFileClose_r:BOOL;
	//bFileRead:BOOL;
	bSave:BOOL;
	bRead:BOOL;
//	tFileOper_Save:TON;
	//tFileOper_Read:TON;
	iDataSetp: INT;
	TON10:Tc2_Standard.TON;
	bExecute: BOOL;
	I1: INT;
	rt100:Tc2_Standard.R_TRIG;
	rt101:Tc2_Standard.R_TRIG;
	bExecute1: BOOL;
	bExecute2: BOOL;
	bExecute3: BOOL;	

	bSaveTemp: BOOL;
	bReadTemp: BOOL;
	bReadDataOk: BOOL;
END_VAR





M_WriteOrRead();

ACTION M_WriteOrRead:



rt100(CLK:=bSave , Q=> );//保存参数
rt101(CLK:=bRead , Q=> );//读取参数

IF rt100.Q THEN
	iDataSetp:=100;
	TON10.IN:=FALSE;
	I1:=1;
	bExecute1:=FALSE;
	bExecute2:=FALSE;	
	bExecute3:=FALSE;	
	bSave:=FALSE;
	bRead:=FALSE;
    bSaveTemp:=TRUE;
	bReadTemp:=FALSE;
END_IF

IF rt101.Q THEN
	iDataSetp:=100;
	TON10.IN:=FALSE;
	I1:=1;
	bExecute1:=FALSE;
	bExecute2:=FALSE;	
	bExecute3:=FALSE;	
	bSave:=FALSE;
	bRead:=FALSE;
    bReadTemp:=TRUE;
    bSaveTemp:=FALSE;
END_IF

TON10(IN:= , PT:=T#200MS , Q=> , ET=> );
//保存配方	
CASE  iDataSetp OF 
	
	100:	//参数给定
	   
	   IF bSaveTemp THEN
	     fbFileOpen_w.nMode:=FOPEN_MODEWRITE OR FOPEN_MODEBINARY;
	   END_IF
	   IF bReadTemp THEN
	     fbFileOpen_w.nMode:=FOPEN_MODEREAD OR  FOPEN_MODEBINARY;
	   END_IF
	  iDataSetp:=101;
	101:

	  CASE I1 OF 
		1:
		 fbFileWrite.pWriteBuff:=ADR(gstM1Par);
		 fbFileWrite.cbWriteLen:=SIZEOF(gstM1Par);
		 fbFileRead.pReadBuff:=ADR(gstM1Par1);
		 fbFileRead.cbReadLen:=SIZEOF(gstM1Par1);
		 fbFileOpen_w.sPathName:='C:\P2Data\M1.csv';//='C:\P2Data\M1.bin';

	  END_CASE
	  iDataSetp:=200;
	
	200:	//打开文件
		bExecute1:=TRUE;
		TON10.IN:=TRUE;
	  IF TON10.Q THEN
		 bExecute1:=FALSE; 
		 TON10.IN:=FALSE;
		 iDataSetp:=300; 
	  END_IF
	
	300:	//读写文件
		bExecute2:=TRUE;
		TON10.IN:=TRUE;
	  IF TON10.Q THEN
		  bExecute2:=FALSE; 
		  TON10.IN:=FALSE;
		 iDataSetp:=400; 
	  END_IF
	
	400:	//关闭文件
		bExecute3:=TRUE;
		TON10.IN:=TRUE;
	  IF TON10.Q THEN
		  bExecute3:=FALSE; 
		  TON10.IN:=FALSE;
		  iDataSetp:=500; 
	  END_IF
	
	500://继续写下个文件
	  IF I1>=1 AND I1<5 THEN
		 I1:=I1+1; 
		 TON10.IN:=FALSE;
		 iDataSetp:=100; 
		 bExecute1:=FALSE; 
		 bExecute2:=FALSE; 
		 bExecute3:=FALSE; 
	  ELSIF I1>=5 THEN
		  bReadTemp:=FALSE;
          bSaveTemp:=FALSE;
		 iDataSetp:=666;   
	  END_IF
END_CASE


IF bReadDataOk THEN
   gstM1Par:=gstM1Par1;
   gstM2Par:=gstM2Par1;
   gstM3Par:=gstM3Par1;
   gstM4Par:=gstM4Par1;	
   gstM5Par:=gstM5Par1;
   bReadDataOk:=FALSE;
END_IF










   	fbFileOpen_w(
	sNetId:= , 
	sPathName:= , //C:\P2Data
	nMode:=   , 
	ePath:=PATH_GENERIC , 
	bExecute:=bExecute1 , 
	tTimeout:=T#3S , 
	bBusy=> , 
	bError=> , 
	nErrId=> , 
	hFile=>hfile );


	fbFileWrite(
	sNetId:= , 
	hFile:= hFile, 
	pWriteBuff:= , 
	cbWriteLen:= , 
	bExecute:=bExecute2 AND bSaveTemp, 
	tTimeout:=T#3S , 
	bBusy=> , 
	bError=> , 
	nErrId=> , 
	cbWrite=> );



	fbFileRead(
	sNetId:= , 
	hFile:=hFile , 
	pReadBuff:= , 
	cbReadLen:= , 
	bExecute:= bExecute2 AND bReadTemp, 
	tTimeout:= T#3S, 
	bBusy=> , 
	bError=> , 
	nErrId=> , 
	cbRead=> , 
	bEOF=> );


	fbFileClose_w(
	sNetId:= , 
	hFile:= hFile, 
	bExecute:= bExecute3, 
	tTimeout:=T#3S , 
	bBusy=> , 
	bError=> , 
	nErrId=> );
END_ACTION

END_FUNCTION_BLOCK

// ---- P2POUs/BasicFunction/08_Data/FB_DataXML_old.TcPOU
FUNCTION_BLOCK FB_DataXML_old
VAR_INPUT
    	bSave:BOOL;
	    bRead:BOOL;
  
END_VAR
VAR_OUTPUT
    	bSaveParDone      :BOOL;
	    bReadParDone     :BOOL;
		bError                     :BOOL;
END_VAR

VAR


	iDataSetp: INT;
	TON10:Tc2_Standard.TON;
	I1: INT;
	rt100:Tc2_Standard.R_TRIG;
	rt101:Tc2_Standard.R_TRIG;
	bExecute1: BOOL;
	bExecute2: BOOL;


	bSaveTemp: BOOL;
	bReadTemp: BOOL;

 fbXmlSrvWrite         : FB_XmlSrvWrite;
// fbXmlSrvWrite         : FB_SrvWrite;
   bExecuteW1             : BOOL;
   sFilePathPar_W       : T_MaxString ;


fbXmlSrvRead   : FB_XmlSrvRead;
//fbXmlSrvRead   : FB_SrvRead;
   bExecuteR          : BOOL;
   sFilePathPar_R      : T_MaxString ;
   sXPathR             : T_MaxString;
	AA: INT;
	BB: INT;












	handleTemp: UDINT;
END_VAR


M_WriteOrRead();

ACTION M_WriteOrRead:
bError := fbXmlSrvWrite.bError OR   fbXmlSrvRead.bError;

rt100(CLK:=bSave , Q=> );//保存参数
rt101(CLK:=bRead , Q=> );//读取参数

IF rt100.Q THEN  //保存参数
	iDataSetp:=100;
	TON10.IN:=FALSE;
	I1:=1;
	bExecute1:=FALSE;
	bExecute2:=FALSE;
	bSave:=FALSE;
	bRead:=FALSE;
    bSaveTemp:=TRUE;
	bReadTemp:=FALSE;
	bSaveParDone:=FALSE;
END_IF

IF rt101.Q THEN  //读取参数
	iDataSetp:=100;
	TON10.IN:=FALSE;
	I1:=1;
	bExecute1:=FALSE;
	bExecute2:=FALSE;	
	bSave:=FALSE;
	bRead:=FALSE;
    bReadTemp:=TRUE;
    bSaveTemp:=FALSE;
	bReadParDone:=FALSE;
END_IF

TON10(IN:= , PT:=T#200MS , Q=> , ET=> );

CASE  iDataSetp OF 
	
 100:
				CASE I1 OF 
				
                 1://轴参数
					sFilePathPar_W  := 'C:\P2XML\P2arrAxisPar.xml';
					fbXmlSrvWrite.pSymAddr:=ADR(arrAxisPar);
					fbXmlSrvWrite.cbSymSize:=SIZEOF(arrAxisPar);   

					sFilePathPar_R  := 'C:\P2XML\P2arrAxisPar.xml';
					fbXmlSrvRead.pSymAddr:=ADR(arrAxisPar);
					fbXmlSrvRead.cbSymSize:=SIZEOF(arrAxisPar);   
                 
				  2://iModeEN
		  		    sFilePathPar_W  := 'C:\P2XML\P2iModeEN.xml';
					fbXmlSrvWrite.pSymAddr:=ADR(iModeEN);
					fbXmlSrvWrite.cbSymSize:=SIZEOF(iModeEN);     

					sFilePathPar_R  := 'C:\P2XML\P2iModeEN.xml';
					fbXmlSrvRead.pSymAddr:=ADR(iModeEN);
					fbXmlSrvRead.cbSymSize:=SIZEOF(iModeEN);   

				  3://P2M1_Par
		  		     sFilePathPar_W  := 'C:\P2XML\P2M1_Par.xml';
					fbXmlSrvWrite.pSymAddr:=ADR(P2M1_Par);
					fbXmlSrvWrite.cbSymSize:=SIZEOF(P2M1_Par);     

					sFilePathPar_R  := 'C:\P2XML\P2M1_Par.xml';
					fbXmlSrvRead.pSymAddr:=ADR(P2M1_Par);
					fbXmlSrvRead.cbSymSize:=SIZEOF(P2M1_Par);   

				  4://P2M2_Par
		  		    sFilePathPar_W  := 'C:\P2XML\P2M2_Par.xml';
					fbXmlSrvWrite.pSymAddr:=ADR(P2M2_Par);
					fbXmlSrvWrite.cbSymSize:=SIZEOF(P2M2_Par);     

					sFilePathPar_R  := 'C:\P2XML\P2M2_Par.xml';
					fbXmlSrvRead.pSymAddr:=ADR(P2M2_Par);
					fbXmlSrvRead.cbSymSize:=SIZEOF(P2M2_Par);   

				  5: //P2M3_Par 
		  		    sFilePathPar_W  := 'C:\P2XML\P2M3_Par.xml';
					fbXmlSrvWrite.pSymAddr:=ADR(P2M3_Par);
					fbXmlSrvWrite.cbSymSize:=SIZEOF(P2M3_Par);     

					sFilePathPar_R  := 'C:\P2XML\P2M3_Par.xml';
					fbXmlSrvRead.pSymAddr:=ADR(P2M3_Par);
					fbXmlSrvRead.cbSymSize:=SIZEOF(P2M3_Par);   
					
				 6: // P2User1_Par
		  		    sFilePathPar_W  := 'C:\P2XML\P2User1_Par.xml';
					fbXmlSrvWrite.pSymAddr:=ADR(P2User1_Par);
					fbXmlSrvWrite.cbSymSize:=SIZEOF(P2User1_Par);     

					sFilePathPar_R  := 'C:\P2XML\P2User1_Par.xml';
					fbXmlSrvRead.pSymAddr:=ADR(P2User1_Par);
					fbXmlSrvRead.cbSymSize:=SIZEOF(P2User1_Par);   					
	
				END_CASE
        IF  bSaveTemp THEN
              handleTemp:=fbXmlSrvWrite.handle;
   	          iDataSetp:=200;
       END_IF
        IF  bReadTemp THEN
              handleTemp:=fbXmlSrvRead.handle;
   	          iDataSetp:=300;
       END_IF

	200:	//保存数据
		bExecute1:=TRUE;
        iDataSetp:=210;
	210:	
       IF  NOT fbXmlSrvWrite.bError  AND NOT fbXmlSrvWrite.bBusy AND handleTemp<>fbXmlSrvWrite.handle  THEN
             iDataSetp:=500;
      END_IF


	300:	//读取参数
		bExecute2:=TRUE;
        iDataSetp:=310;
	310:	
       IF  NOT fbXmlSrvRead.bError  AND NOT fbXmlSrvRead.bBusy AND handleTemp<>fbXmlSrvRead.handle  THEN
             iDataSetp:=500;
      END_IF


	500://继续写下个文件
	  IF I1>=1 AND I1<6 THEN
		 I1:=I1+1; 
		 iDataSetp:=100; 
		 bExecute1:=FALSE; 
		 bExecute2:=FALSE; 
	  ELSIF I1>=6 THEN
          IF  bSaveTemp THEN
               bSaveParDone:=TRUE;
         END_IF

          IF  bReadTemp THEN
               bReadParDone:=TRUE;
         END_IF

		  bReadTemp:=FALSE;
          bSaveTemp:=FALSE;

	   	 iDataSetp:=666;   
	  END_IF
END_CASE


AA:=BB;

fbXmlSrvWrite(
   nMode           := XMLSRV_ADDMISSING,
   pSymAddr        :=,//ADR(Value1)
   cbSymSize       := ,//SIZEOF(Value1)
   sFilePath       := sFilePathPar_W,
   sXPath	       := '/dataentry/value',
   bExecute        := bExecute1
);


fbXmlSrvRead(
   pSymAddr       := ,
   cbSymSize      := ,
   sFilePath      := sFilePathPar_R,
   sXPath	         := '/dataentry/value',
   bExecute       := bExecute2
);
END_ACTION

END_FUNCTION_BLOCK

// ---- P2POUs/BasicFunction/09_User1/Dp_Roll_New_BAK.TcPOU
FUNCTION_BLOCK Dp_Roll_New_BAK
VAR_IN_OUT
	AxisM:AXIS_REF;//旋转虚轴
	Axis_P:AXIS_REF;//平移轴
	Axis_S:AXIS_REF;//升降轴
	JuanRao_PY:ARRAY[0..MaxNo] OF sMC_CAM_REF;
	JuanRao_SJ:ARRAY[0..MaxNo] OF sMC_CAM_REF;
END_VAR
VAR_INPUT
	Enable:BOOL;
	Width:REAL;//电芯宽度
	Thick:REAL;//电芯厚度
	r1:REAL;//电芯转角-圆角半径
END_VAR
VAR_OUTPUT
	Enabling:BOOL;
	Done:BOOL;
	Busy:BOOL;
	Alm:BOOL;
END_VAR
VAR
	Enable_R: R_TRIG;
	Enable_F: F_TRIG;
	TON1: TON;
	P_Off: BOOL;
	// 初始倒角圆心坐标X0
	Circle_X0: LREAL;
	// 初始倒角圆心坐标Y0
	Circle_Y0: LREAL;
	// 初始切点坐标X0
	QieDian_X0: LREAL;
	// 初始切点坐标Y0
	QieDian_Y0: LREAL;
	// 初始倒角圆心负角度
	Circle_Angle0: LREAL;
	// 初始倒角圆心负角度的右侧角度
	MidAngle: LREAL;
	// 90度左侧倒角圆切点到中心的角度
	QieDian_Angle90: LREAL;
	// 初始切点到中心的上角度
	QieDian_AngleUp: LREAL;
	// 初始切点到中心的下角度
	QieDian_AngleDn: LREAL;
	// 初始圆角切点至中心距离
	Circle_Line0: LREAL;
	// 初始圆角切点至中心距离
	QieDian_Line0: LREAL;
	i: INT;
	// 实时倒角圆心坐标x1
	C_X: LREAL;
	// 实时倒角圆心坐标y1
	C_Y: LREAL;
	// 实时倒角圆心坐标x2
	Q_X: LREAL;
	// 实时切点圆心坐标x
	Q_Y: LREAL;
	// 圆弧对应的角度
	Arc_Angle: LREAL;
	// 圆弧对应的弧长
	Arc_Len: LREAL;
	New3_Scale_FB: ARRAY[1..4] OF New3_Scale;
	// 升降轴运动长度/mm
	AxisYmm: LREAL;
	// 平移轴运动长度/mm
	AxisXmm: LREAL;
	OUT1: LREAL;
	// 90度后切点的角度
	QieDian_Angle: LREAL;
END_VAR
VAR CONSTANT
	MaxNo: INT := 360;//凸轮数据索引常量
	Pai: LREAL := 3.1415926535;
END_VAR

Enable_R(CLK:=Enable);Enable_F(CLK:=Enable);
Enabling:=Enable;
//Pai:=3.1415926535;
(*前提条件：XY坐标系，电芯旋转中心坐标为(0,0)，电芯模型四个角为圆角，半径r1*)
IF Enable_F.Q THEN
	TON1(IN:=P_Off,PT:=T#100ms);
	Busy:=FALSE;Alm:=FALSE;
	Done:=FALSE;
END_IF;
IF Enable_R.Q  AND (NOT Busy) AND (NOT Alm)THEN
	Busy:=TRUE;Alm:=FALSE;Done:=FALSE;
END_IF;
IF Enable AND Busy THEN		
	IF Thick*0.5-r1<0 THEN
		Alm:=TRUE;(*圆角半径尺寸错误*)
		RETURN;
	END_IF;
	Circle_X0:=-Width*0.5+r1;			(*初始离切点最近的圆心坐标，该点在中心左侧，负数*)
	Circle_Y0:=Thick*0.5-r1;				(*初始离切点最近的圆心坐标，该点在中心上方，正数*)

	QieDian_X0:=-Width*0.5+r1;		(*初始切点坐标，该点在中心左侧，负数*)
	QieDian_Y0:=Thick*0.5;				(*初始切点坐标，该点在中心上方，正数*)	

	Circle_Angle0:=(180*ATAN(Circle_Y0/Circle_X0))/Pai;  (*负角度*)
	MidAngle:=180+Circle_Angle0;     (*-X轴角度是180°*)		

	QieDian_Angle90:=(180*ATAN(-Circle_Y0/(Width*0.5)))/Pai;		(*负角度*)

	QieDian_AngleUp:=(180*ATAN(QieDian_Y0/QieDian_X0))/Pai;	(*负角度*)
	QieDian_AngleDn:=(180*ATAN(-QieDian_Y0/QieDian_X0))/Pai;	(*正角度*)		
	
	Circle_Line0:=SQRT(Circle_X0*Circle_X0+Circle_Y0*Circle_Y0);
	QieDian_Line0:=SQRT(QieDian_X0*QieDian_X0+QieDian_Y0*QieDian_Y0);

	JuanRao_PY[0].Phase:=0;JuanRao_PY[0].Distance:=0;	
	JuanRao_SJ[0].Phase:=0;JuanRao_SJ[0].Distance:=0;

	FOR i:=1 TO 360 BY 1 DO
		MidAngle:=MidAngle-0.5;
		IF (i<=180) THEN
			C_X:=Circle_Line0*COS((MidAngle)*Pai/180);							(*初始倒角圆心运动中的X坐标*)
			C_Y:=Circle_Line0*SIN((MidAngle)*Pai/180);							(*初始倒角圆心运动中的Y坐标*)
			Q_X:=QieDian_Line0*COS((180+QieDian_AngleUp-INT_TO_REAL(i)/2)*Pai/180);				(*初始切点运动中的X坐标*)
			Q_Y:=QieDian_Line0*SIN((180+QieDian_AngleUp-INT_TO_REAL(i)/2)*Pai/180);				(*初始切点运动中的Y坐标*)
			Arc_Angle:=90-(180*ATAN((Q_Y-C_Y)/(Q_X-C_X)))/Pai;		(*圆弧对应的夹角:=90-两圆心的夹角*)
			Arc_Len:=Arc_Angle*Pai*r1/180;											(*由圆弧的夹角求出弧长*)		
			New3_Scale_FB[1](X:=INT_TO_REAL(i) , Sall:= Width*0.5-Thick*0.5, T:=180 , OUT=>AxisYmm );
			AxisXmm:=C_X-Circle_X0+Arc_Len;
			IF i=180 THEN
				QieDian_Line0:=SQRT(Circle_Y0*Circle_Y0+Width*0.5*Width*0.5);  (*切点变了*)
			END_IF;
		ELSE 			
			C_X:=Circle_Line0*COS((MidAngle-2*Circle_Angle0)*Pai/180);(*注意切点从前倒角变成后倒角*)
			C_Y:=Circle_Line0*SIN((MidAngle-2*Circle_Angle0)*Pai/180);
			QieDian_Angle:=180-INT_TO_REAL(i)/2-QieDian_Angle90;
			Q_X:=QieDian_Line0*COS(QieDian_Angle*Pai/180);
			Q_Y:=QieDian_Line0*SIN(QieDian_Angle*Pai/180);
			Arc_Angle:=90-(180*ATAN((Q_Y-C_Y)/(Q_X-C_X)))/Pai;
			Arc_Len:=Arc_Angle*Pai*r1/180;
			New3_Scale_FB[3](X:=INT_TO_REAL(i)-180 , Sall:=Width*0.5-(Thick*0.5), T:=180 , OUT=>OUT1 );
			AxisYmm:=Width*0.5-(Thick*0.5)-OUT1;
			AxisXmm:=C_X-QieDian_X0+Arc_Len+(Thick-2*r1+Pai*r1*0.5);(*水平位置*)
		END_IF;	
		JuanRao_PY[i].Phase:=INT_TO_REAL(i)/2;	JuanRao_PY[i].Distance:=LREAL_TO_REAL(AxisXmm);				
		JuanRao_SJ[i].Phase:=INT_TO_REAL(i)/2;		JuanRao_SJ[i].Distance:=LREAL_TO_REAL(AxisYmm);		
		IF  i=360 THEN 
			JuanRao_SJ[i].Distance:=0;
		END_IF;
	END_FOR;
	Done:=TRUE;Busy:=FALSE;	
(*
	TON1(IN:=Busy,PT:=T#100ms);
	MC_CamIn_ROLL[1](Master:=AxisM, Slave:=Axis_P, CamTable:=JuanRao_PY, Execute:=TON1.Q, Periodic:=TRUE,StartMode:=_mcRelativePosition,StartPosition:=AxisM.Act.Pos,SlaveOffset:=0);
	MC_CamIn_ROLL[2](Master:=AxisM, Slave:=Axis_S, CamTable:=JuanRao_SJ, Execute:=TON1.Q, Periodic:=TRUE,StartMode:=_mcRelativePosition,StartPosition:=AxisM.Act.Pos,SlaveOffset:=0);
	IF TON1.Q THEN
		Done:=TRUE;Busy:=FALSE;	
	END_IF;
*)	
END_IF;

END_FUNCTION_BLOCK

// ---- P2POUs/BasicFunction/09_User1/Dp_Roll_V2.TcPOU
FUNCTION_BLOCK Dp_Roll_V2
VAR_IN_OUT
   	Enable:BOOL;
   
END_VAR

VAR_INPUT
    fAngleRel:LREAL;//电芯旋转角度
	Width:REAL;//电芯宽度
	Thick:REAL;//电芯厚度
	 r0:    REAL;//   隔膜夹板初始位置到电芯 初始位置A点距离
	
	
	//r1:REAL;//电芯转角-圆角半径
END_VAR
VAR_OUTPUT

END_VAR

VAR_IN_OUT
	iMode: INT;
END_VAR
VAR
	Enable_R: R_TRIG;
	Enable_F: F_TRIG;
	TON1: TON;
	P_Off: BOOL;
	// 初始倒角圆心坐标X0
	Circle_X0: LREAL;
	// 初始倒角圆心坐标Y0
	Circle_Y0: LREAL;
	// 初始切点坐标X0
	QieDian_X0: LREAL;
	// 初始切点坐标Y0
	QieDian_Y0: LREAL;
	// 初始倒角圆心负角度
	Circle_Angle0: LREAL;
	// 初始倒角圆心负角度的右侧角度
	MidAngle: LREAL;
	// 90度左侧倒角圆切点到中心的角度
	QieDian_Angle0: LREAL;
	// 初始切点到中心的上角度
	QieDian_AngleUp: LREAL;
	// 初始切点到中心的下角度
	QieDian_AngleDn: LREAL;
	// 初始圆角切点至中心距离
	Circle_Line0: LREAL;
	// 初始圆角切点至中心距离
	QieDian_Line0: LREAL;
	i: INT;
	// 实时倒角圆心坐标x1
	C_X: LREAL;
	// 实时倒角圆心坐标y1
	C_Y: LREAL;
	// 实时倒角圆心坐标x2
	Q_X: LREAL;
	// 实时切点圆心坐标x
	Q_Y: LREAL;
	// 圆弧对应的角度
	Arc_Angle: LREAL;
	// 圆弧对应的弧长
	Arc_Len: LREAL;
	//New3_Scale_FB: ARRAY[1..4] OF New3_Scale;
	// 升降轴运动长度/mm
	AxisYmm: LREAL;
	// 平移轴运动长度/mm
	AxisXmm: LREAL;
	OUT1: LREAL;
	// 90度后切点的角度
	QieDian_Angle: LREAL;
	MA1: BOOL;
	Circle_X1: LREAL;
	Circle_Y1: LREAL;
	QieDian_X1: LREAL;
	QieDian_Y1: REAL;
	Circle_Angle1: LREAL;
	QieDian_Angle1: LREAL;
	Circle_Line1: LREAL;
	QieDian_Line1: LREAL;
	
	
	JiaoDianA_X0:LREAL;
	JiaoDianA_Y0:LREAL;	
	JiaoDian_Angle0: LREAL; //
	JiaoDian_Line0: LREAL; //
	
  	 GMBoard_X0:LREAL;  
	 GMBoard_Y0:LREAL;  
	 
	r1: REAL;	 
	r2: REAL;
	r3: REAL;
	
	 JDA_X: LREAL;
	 JDA_Y: LREAL;
	 JDB_X: LREAL;
	 JDB_Y: LREAL;	
	 JDC_X: LREAL;
	 JDC_Y: LREAL;		 
	 JDD_X: LREAL;
	 JDD_Y: LREAL;		 
	 
	 
	
	a: LREAL;
	b: REAL;
	JDX: LREAL;
	c: LREAL;
	JDY: LREAL;
	RJD: LREAL;
	fResult: LREAL;
	fResult1: LREAL;
	fDelta: LREAL;
	fResult2: LREAL;
	bError: BOOL;
	bCacleOnce: BOOL;
	bError2: BOOL;
	bMA1: BOOL;

	k: REAL;
	fAngleRelTemp1: LREAL;
	fAngleRelTemp2: LREAL;
	fAngleRelTemp3: LREAL;
	bTest: BOOL;
	iFLG1: INT;
END_VAR
VAR CONSTANT
	MaxNo: INT := 360;//凸轮数据索引常量
	Pai: LREAL := 3.1415926535;
END_VAR


Enable_R(CLK:=Enable);Enable_F(CLK:=Enable);

IF Enable_F.Q THEN
	TON1(IN:=P_Off,PT:=T#100MS);
END_IF;

IF Enable   THEN		
		IF Thick*0.5<0 THEN
	
			RETURN;
		 END_IF;
	
			  AxisXmm:=0;
			  AxisYmm:=0;
			  Arc_Angle:=0;		    
			  Arc_Len:=0;			
	///SJ
	  JiaoDianA_X0:=-Width*0.5;
	  JiaoDianA_Y0:= Thick*0.5;
	  JiaoDian_Angle0:=ABS( (180*ATAN(JiaoDianA_Y0/JiaoDianA_X0))/Pai )  ;  (*初始圆心角度*)
	 // Circle_Line0:=SQRT(Circle_X0*Circle_X0+Circle_Y0*Circle_Y0);
	  JiaoDian_Line0:=SQRT(JiaoDianA_X0*JiaoDianA_X0+JiaoDianA_Y0*JiaoDianA_Y0);
	  
	  GMBoard_X0:=-Width*0.5-r0;
	  GMBoard_Y0:=  Thick*0.5;
	  
	  r1:=r0-Width;
	  r2:=r0-Width-Thick;
	  r3:=r0-Width-Thick-Width;

  

	//A点到F点 距离=ro     (JDA_X-x )* (JDA_X-x )+(JDA_Y-GMBoard_Y0)*(JDA_Y-GMBoard_Y0)=r0*r0
	
	  IF   JiaoDian_Angle0 -fAngleRel>=0 THEN    //A  点在第一象限    A点半径  r0
			   JDA_X:=-JiaoDian_Line0*COS((JiaoDian_Angle0 -fAngleRel)*Pai/180);	//A
			   JDA_Y:=JiaoDian_Line0*SIN((JiaoDian_Angle0 -fAngleRel)*Pai/180);		
			   //解方程
			   JDX:=JDA_X;
			   JDY:=JDA_Y;
			   RJD:=r0;
			   bCacleOnce:=TRUE;	   
	 ELSIF   fAngleRel -JiaoDian_Angle0>0		AND    fAngleRel -JiaoDian_Angle0<=90 THEN    //A  点在第e二象限    A点半径  r0 
				JDA_X:=-JiaoDian_Line0*COS((fAngleRel -JiaoDian_Angle0)*Pai/180);
				JDA_Y:=-JiaoDian_Line0*SIN((fAngleRel -JiaoDian_Angle0)*Pai/180);		
			   //解方程
			   JDX:=JDA_X;
			   JDY:=JDA_Y;
			   RJD:=r0;
			   bCacleOnce:=TRUE;	   	   
				   
	 ELSIF  180+JiaoDian_Angle0-fAngleRel >=0     AND     180+JiaoDian_Angle0-fAngleRel <90 THEN    //A  点在第三象限   判断D点的位置  如果                                  A点半径  r0 		   
				JDA_X:=JiaoDian_Line0*COS((180+JiaoDian_Angle0-fAngleRel)*Pai/180);
				JDA_Y:=-JiaoDian_Line0*SIN((180+JiaoDian_Angle0-fAngleRel)*Pai/180);	
			   
			   //判断D点是在第一象限还是在二象限
			   IF 180-JiaoDian_Angle0-fAngleRel<=90 AND   180-JiaoDian_Angle0-fAngleRel>=0    THEN   //一象限
					 JDD_X:=-JiaoDian_Line0*COS((180-JiaoDian_Angle0-fAngleRel)*Pai/180);
					 JDD_Y:= JiaoDian_Line0*SIN((180-JiaoDian_Angle0-fAngleRel)*Pai/180);	
					 
			   ELSIF  fAngleRel-(180- JiaoDian_Angle0 ) >0 AND  fAngleRel-(180- JiaoDian_Angle0 ) <=90 THEN     //二象限
					 JDD_X:=-JiaoDian_Line0*COS((  fAngleRel-(180- JiaoDian_Angle0 ) )*Pai/180);
					 JDD_Y:=-JiaoDian_Line0*SIN((  fAngleRel-(180- JiaoDian_Angle0 )   )*Pai/180);		
	    		   
			   END_IF
			   
	   
			   //判断D点是在直线AF 上方还是直线下方 
			   IF   iMode=1 THEN   // 先计算一次
					 JDX:=JDA_X;
					 JDY:=JDA_Y;
					 RJD:=r0;
					 bCacleOnce:=TRUE;	
					// iMode:=1;   	   
			   END_IF
			   
			   IF     iMode=2  THEN   //        
					 JDX:=JDD_X;
					 JDY:=JDD_Y;
					 RJD:=r1;
					 bCacleOnce:=TRUE;	
			   END_IF		   
	
	ELSIF     fAngleRel -JiaoDian_Angle0-180>0  AND     fAngleRel -JiaoDian_Angle0-180<=90  THEN                                                   //A  点在第四象限   
			   //判断D点是在第二象限还是在三象限
			   IF  fAngleRel-(180- JiaoDian_Angle0 ) >=0 AND  fAngleRel-(180- JiaoDian_Angle0 ) <=90 THEN     //二象限
					 JDD_X:=-JiaoDian_Line0*COS((  fAngleRel-(180- JiaoDian_Angle0 ) )*Pai/180);
					 JDD_Y:=-JiaoDian_Line0*SIN((  fAngleRel-(180- JiaoDian_Angle0 )   )*Pai/180);		
			   ELSIF  360-fAngleRel-JiaoDian_Angle0 >=0    AND  360-fAngleRel-JiaoDian_Angle0 <90   THEN     //三象限
					 JDD_X:=JiaoDian_Line0*COS(( 360-fAngleRel-JiaoDian_Angle0  )*Pai/180);
					 JDD_Y:=-JiaoDian_Line0*SIN((  360-fAngleRel-JiaoDian_Angle0   )*Pai/180);			    		   
			   END_IF
			   
			   //判断C点是在第一象限还是在二象限(   C点只能在第2象限     )
					 JDC_X:=-JiaoDian_Line0*COS((  fAngleRel -JiaoDian_Angle0-180)*Pai/180);
					 JDC_Y:=-JiaoDian_Line0*SIN((  fAngleRel -JiaoDian_Angle0-180)*Pai/180);			   
	
				   //判断C点是在直线DF 上方还是直线下方 
			   IF    iMode=2 THEN   // 先计算一次
					 JDX:=JDD_X;
					 JDY:=JDD_Y;
					 RJD:=r1;
					 bCacleOnce:=TRUE;	
					// iMode:=3;   	   
			   END_IF
			   
			   IF    iMode=4  THEN   //        
					 JDX:=JDC_X;
					 JDY:=JDC_Y;
					 RJD:=r2;
					 bCacleOnce:=TRUE;	
			   END_IF		   	   
			
	ELSIF  360- fAngleRel + JiaoDian_Angle0 >=0   AND 360- fAngleRel + JiaoDian_Angle0 <90 THEN           //A  点在第1象限   
			   //判断C点是在第一象限还是在二象限(   C点只能在第3象限     )
				 JDC_X:=JiaoDian_Line0*COS((  360-fAngleRel+JiaoDian_Angle0)*Pai/180);
				 JDC_Y:=-JiaoDian_Line0*SIN((  360-fAngleRel+JiaoDian_Angle0)*Pai/180);	
	
			   //判断B点是在第1象限还是在2象限
			   IF   360-fAngleRel-JiaoDian_Angle0 >=0 AND   360-fAngleRel-JiaoDian_Angle0 <=90 THEN     //1象限
					 JDB_X:=-JiaoDian_Line0*COS((  360-fAngleRel-JiaoDian_Angle0 )*Pai/180);
					 JDB_Y:= JiaoDian_Line0*SIN((   360-fAngleRel-JiaoDian_Angle0  )*Pai/180);		
					 iFLG1:=1;
			   ELSIF  JiaoDian_Angle0-( 360- fAngleRel ) >0    AND  JiaoDian_Angle0-( 360- fAngleRel )<=90   THEN     //2象限
					 JDB_X:= -JiaoDian_Line0*COS(( JiaoDian_Angle0-( 360- fAngleRel )  )*Pai/180);
					 JDB_Y:= - JiaoDian_Line0*SIN((  JiaoDian_Angle0-( 360- fAngleRel )    )*Pai/180);			 
   		              iFLG1:=2;
			   END_IF
		   
				   //判断C点是在直线DF 上方还是直线下方 
			   IF    iMode=4 THEN   // 先计算一次
					 JDX:=JDC_X;
					 JDY:=JDC_Y;
					 RJD:=r2;
					 bCacleOnce:=TRUE;	
				//	 iMode:=5;   	   
			   END_IF
			   
			   IF    iMode=6  THEN   //        
					 JDX:=JDB_X;
					 JDY:=JDB_Y;
					 RJD:=r3;
					 bCacleOnce:=TRUE;	
			   END_IF		 
	
	 END_IF
  
  
  
	  //解一元二次方程   JDX : 当前圆心X      JDY:当前圆心Y     RJD: 当前圆心半径
	  //    (JDX-x )* (X-x )+(JDY-GMBoard_Y0)*(JDY-GMBoard_Y0)=RJD*RJD 
	IF bCacleOnce  THEN  
			  a:=1;
			  b:=-2*JDX;
			  c:=JDX*JDX+(JDY-GMBoard_Y0)*(JDY-GMBoard_Y0)-RJD*RJD;
			  
			  fDelta:=b*b-4*a*c;
			  
			  IF  fDelta>=0 THEN
				  fResult1:= (-b+SQRT(fDelta) )/ (2*a);
				  fResult2:= (-b-SQRT(fDelta) )/ (2*a);
			ELSE	  
				  ;
			 END_IF
			  
			IF fDelta>=0 THEN  
				  IF fResult1<fResult2 THEN
					  fResult:=fResult1;
				  ELSE 
					  fResult:=fResult2;  
				  END_IF
			ELSE
			  // fResult:=0;  
			   bError:=TRUE;
			END_IF  
		 bCacleOnce:=FALSE;
		
	END_IF 
  
//  IF NOT  bCacleOnce AND   Enable AND  NOT  bError     THEN 
 IF NOT  bCacleOnce AND   Enable      THEN
		 AxisXmm:=fResult-GMBoard_X0;  //X位移变化
		 
		 IF iMode=1  AND  180+JiaoDian_Angle0-fAngleRel >=0  AND     180+JiaoDian_Angle0-fAngleRel <90    THEN   //判断点D  相对与直线AF 的位置
			 k:= (JDA_Y-GMBoard_Y0)/( JDA_X- fResult );
		     b:= JDA_Y-k*JDA_X;
		    //将 D点代入  直线AF   
		    IF k*JDD_X+b <JDD_Y THEN  //D点在直线 AF上方
				 bMA1:=FALSE;
			ELSIF  k*JDD_X+b =JDD_Y THEN ////D点在直线 AF上
			     bMA1:=FALSE;
			ELSIF  k*JDD_X+b >JDD_Y THEN
			     bMA1:=TRUE;
				  fAngleRelTemp1:= fAngleRel;
				  iMode:=2;
			END_IF
		 END_IF
		 
		 IF iMode=2 AND  fAngleRel -JiaoDian_Angle0-180>0  AND     fAngleRel -JiaoDian_Angle0-180<=90   THEN   //判断点C  相对与直线DF 的位置
			 k:= (JDD_Y-GMBoard_Y0)/( JDD_X- fResult );
		     b:= JDD_Y-k*JDD_X;
		    //将 C点代入  直线AF   
		    IF k*JDC_X+b <JDC_Y THEN  //D点在直线 AF上方
				 bMA1:=FALSE;
			ELSIF  k*JDC_X+b =JDC_Y THEN ////D点在直线 AF上
			     bMA1:=FALSE;
			ELSIF  k*JDC_X+b >JDC_Y THEN
			     bMA1:=TRUE;
				  fAngleRelTemp2:= fAngleRel;
				  iMode:=4;
			END_IF
		 END_IF		 
		 
		 IF iMode=4 AND   360- fAngleRel + JiaoDian_Angle0 >=0   AND 360- fAngleRel + JiaoDian_Angle0 <90   THEN   //判断点B  相对与直线CF 的位置
			 k:= (JDC_Y-GMBoard_Y0)/( JDC_X- fResult );
		     b:= JDC_Y-k*JDC_X;
		    //将 B点代入  直线CF  
		    IF k*JDB_X+b <JDB_Y THEN  //D点在直线 AF上方
				 bMA1:=FALSE;
			ELSIF k*JDB_X+b =JDB_Y THEN ////D点在直线 AF上
			     bMA1:=FALSE;
			ELSIF  k*JDB_X+b >JDB_Y THEN
			     bMA1:=TRUE;
				   fAngleRelTemp3:= fAngleRel;
				  iMode:=6;
			END_IF
		 END_IF		 
		
	    Enable:=FALSE;	 
ELSE
	 bError2:=TRUE;	  //无触发计算
END_IF
  
  

END_IF






	IF bTest        THEN  
			  a:=1;
			  b:=-2*JDX;
			  c:=JDX*JDX+(JDY-GMBoard_Y0)*(JDY-GMBoard_Y0)-RJD*RJD;
			  
			  fDelta:=b*b-4*a*c;
			  
			  fResult1:= (-b+SQRT(fDelta) )/ (2*a);
			  fResult2:= (-b-SQRT(fDelta) )/ (2*a);
			  
			IF fDelta>0 THEN  
				  IF fResult1<fResult2 THEN
					  fResult:=fResult1;
				  ELSE 
					  fResult:=fResult2;  
				  END_IF
			ELSE
			   fResult:=0;  
			   bError:=TRUE;
			END_IF  
		 bTest:=FALSE;
		
	END_IF

END_FUNCTION_BLOCK

// ---- P2POUs/BasicFunction/09_User1/FB_CrectCamYaDaoLine.TcPOU
FUNCTION_BLOCK FB_CrectCamYaDaoLine	
VAR_INPUT
   	bCreatTable		                         :BOOL;	
	Reset                                        :BOOL;  
	iTable		                                :UINT;    


    fMoveLength                                 :REAL:=40;   //压倒平移最大距离
    
    fMasterKeyPos1                           :REAL:=164;   
    fMasterKeyPos2                           :REAL:=241;   
    fMasterKeyPos3                           :REAL:=289;  
    fMasterKeyPos4                           :REAL:=289;  
	 
	fMoveLength2                             :REAL:=-15;   //压刀压隔膜长度
END_VAR

VAR_IN_OUT
	axisSlave		                            :axis_ref;  
	axisMaster		                            :axis_ref;  
END_VAR

VAR_OUTPUT
    bCreatTableDone                        :BOOL;
    bCreatTableError                        :BOOL;
	bError                         :BOOL;

END_VAR


VAR
	rtrigs		                                      :ARRAY[1..3]OF R_TRIG;
	ftrigs		                                      :ARRAY[1..3]OF F_TRIG;
    PositionData1			                  :ARRAY[1..6] OF MC_MotionFunctionPoint;	////
	fbCamtableselect:		               	MC_CamTableSelect;////
	Cam_table:				MC_CAM_REF;////
	bWriteCamData: BOOL;
    iCreatTableStep       :INT;
END_VAR


rtrigs[1](CLK:=bCreatTable);  
ftrigs[1](CLK:=bCreatTable);  

CASE iCreatTableStep OF   
0:  
    IF  rtrigs[1].Q  AND NOT bCreatTableError  THEN
         fbCamtableselect.Execute:=FALSE;
         bCreatTableDone:=FALSE;
         bCreatTable:=FALSE;
         bWriteCamData:=TRUE;
         iCreatTableStep:=10;
    END_IF 

10: 
   IF NOT bWriteCamData THEN 
	  fbCamtableselect.Execute:=TRUE;   
	 iCreatTableStep:=20;	
  END_IF

20:		
	IF NOT  fbCamtableselect.Execute   THEN
        bCreatTableDone:=TRUE;
		iCreatTableStep:=0;	
    ELSIF  fbCamtableselect.Error        THEN
       bCreatTableError:=TRUE;
       iCreatTableStep:=999;	//创建凸轮失败
	END_IF		
END_CASE

(**********故障***********)
	IF  Reset  AND bCreatTableError  THEN  
	   bCreatTableError:=FALSE;
	   iCreatTableStep:=0;
	END_IF


ModifyCam();

ACTION ModifyCam:

fbCamtableselect(   
	Execute:=                        fbCamtableselect.Execute ,
	Periodic:=                        FALSE ,
	MasterAbsolute:=             FALSE,
	SlaveAbsolute:=                FALSE ,
	CamTableID:=                  iTable,
	Master:=                         axisMaster ,
	Slave:=                            axisSlave ,
	CamTable:=                     Cam_table , );

IF fbCamtableselect.Done THEN
    fbCamtableselect.Execute:=FALSE;
END_IF

IF bWriteCamData  THEN

	  Cam_table.ArraySize:=SIZEOF(PositionData1); 
	  Cam_table.NoOfColumns:=1;
	  Cam_table.NoOfRows:=6;
	  Cam_table.pArray:=ADR(PositionData1);
	  Cam_table.TableType:=MC_TABLETYPE_MOTIONFUNCTION;
  
      //MOTIONFUNCTYPE_BESCHLTRAPEZ     MOTIONFUNCTYPE_POLYNOM7_MM    MOTIONFUNCTYPE_BESCHLTRAPEZ   MOTIONFUNCTYPE_POLYNOM1

	  PositionData1[1].	PointIndex	:=	        1;
	  PositionData1[1].	FunctionType	:=		MOTIONFUNCTYPE_POLYNOM1;
	  PositionData1[1].	PointType	:=	        MOTIONPOINTTYPE_MOTION;
	  PositionData1[1].	RelIndexNextPoint	:=  1;
	  PositionData1[1].	MasterPos	:=	        0;
	  PositionData1[1].	SlavePos	:=	        0;		//fMoveLength
	  PositionData1[1].	SlaveVelo	:=	        0;
	  
	  PositionData1[2].	PointIndex	:=	        2;
	  PositionData1[2].	FunctionType	:=		MOTIONFUNCTYPE_POLYNOM5_MM;
	  PositionData1[2].	PointType	:=	        MOTIONPOINTTYPE_MOTION;
	  PositionData1[2].	RelIndexNextPoint	:=  1;
	  PositionData1[2].	MasterPos	:=	        fMasterKeyPos1;
	  PositionData1[2].	SlavePos	:=	        0;	
	  PositionData1[2].	SlaveVelo	:=	        0	;

	  PositionData1[3].	PointIndex	:=	        3;
	  PositionData1[3].	FunctionType	:=		MOTIONFUNCTYPE_POLYNOM5_MM;
	  PositionData1[3].	PointType	:=	        MOTIONPOINTTYPE_MOTION;
	  PositionData1[3].	RelIndexNextPoint	:=  1;
	  PositionData1[3].	MasterPos	:=	        fMasterKeyPos4;
	  PositionData1[3].	SlavePos	:=	        fMoveLength2;	//-15
	  PositionData1[3].	SlaveVelo	:=	        -1	;  
	  
	  PositionData1[4].	PointIndex	:=	        4;
	  PositionData1[4].	FunctionType	:=		MOTIONFUNCTYPE_POLYNOM5_MM;
	  PositionData1[4].	PointType	:=	        MOTIONPOINTTYPE_MOTION;
	  PositionData1[4].	RelIndexNextPoint	:=  0;
	  PositionData1[4].	MasterPos	:=	        fMasterKeyPos2;
	  PositionData1[4].	SlavePos	:=	        fMoveLength;	
	  PositionData1[4].	SlaveVelo	:=	        0	;

	  PositionData1[5].	PointIndex	:=	        5;
	  PositionData1[5].	FunctionType	:=		MOTIONFUNCTYPE_POLYNOM1;
	  PositionData1[5].	PointType	:=	        MOTIONPOINTTYPE_MOTION;
	  PositionData1[5].	RelIndexNextPoint	:=  1;
	  PositionData1[5].	MasterPos	:=	        fMasterKeyPos3;//fMasterKeyPos
	  PositionData1[5].	SlavePos	:=	        0;	
	  PositionData1[5].	SlaveVelo	:=	       0	;

	  PositionData1[6].	PointIndex	:=	        6;
	  PositionData1[6].	FunctionType	:=		MOTIONFUNCTYPE_POLYNOM1;
	  PositionData1[6].	PointType	:=	        MOTIONPOINTTYPE_MOTION;
	  PositionData1[6].	RelIndexNextPoint	:=  0;
	  PositionData1[6].	MasterPos	:=	        360;
	  PositionData1[6].	SlavePos	:=	        0;	
	  PositionData1[6].	SlaveVelo	:=	       0	;

     bWriteCamData:=FALSE;
END_IF
END_ACTION

END_FUNCTION_BLOCK

// ---- P2POUs/BasicFunction/10_MES/CS_CcdTcp.TcPOU
FUNCTION_BLOCK PUBLIC CS_CcdTcp
VAR_INPUT
END_VAR
VAR_OUTPUT
END_VAR
VAR_IN_OUT
   iCcd2:ICCD;
   Data:STCcdData;
END_VAR


VAR
	ccdDataSend:STCcdDataSend;
	
	fbTcpCon:FB_SocketConnect;
	fbTcpSend:FB_SocketSend;
	fbTcpRec:FB_SocketReceive;
	fbTcpClose: FB_SocketClose;
	bConnect: BOOL;
	bClose: BOOL;
	hTcpSock: T_HSOCKET;
	//aTcpSend:ARRAY[1..10] OF BYTE;
	//aTcpReceive:ARRAY[1..10] OF BYTE;	
	StrSend:STRING;
	StrReceive:STRING;
	fbUdpCreate:FB_SocketUdpCreate;
	hUdp: T_HSOCKET;
	bCreate: BOOL;
	port: UDINT:=9004;
	bSendTcp: BOOL;
	bReceiveTcp: BOOL;
	fbSwingHalt2: MC_Halt;



END_VAR




	Config();
	
	M_SendReceive();


	
	

	
	
	
	

	
	
	
	
	
	
	
	
	
	
	
	
	
	
	
	
	
(*	
   fbUdpCreate(
	sSrvNetId:= , 
	sLocalHost:= , 
	nLocalPort:= port, 
	bExecute:=bCreate , 
	tTimeout:= , 
	bBusy=> , 
	bError=> , 
	nErrId=> , 
	hSocket=> hUdp);
	
	
	*)

ACTION Config:



  IF iCcd2.bComOpen THEN
	 bConnect:=TRUE;	
	 bClose:=FALSE;
	 iCcd2.bComOpen:=FALSE;
  END_IF
  
   IF iCcd2.bComClose THEN
	 bConnect:=FALSE;	
	 bClose:=TRUE;
	 iCcd2.bComClose:=FALSE;
  END_IF 
  
  
  //第一步，编写 TCP/IP 连接功能块
fbTcpCon(
	sSrvNetId:= ''   ,          //       (*'169.254.46.193.1.1'*) , 
	sRemoteHost:='192.168.2.11'     , 
	nRemotePort:= 2020, //端口号；
	bExecute:=bConnect , //连接执行位；
	tTimeout:= , 
	bBusy=> , 
	bError=> , 
	nErrId=> , 
	hSocket=>hTcpSock );
	
	
//第四步，编写 TCP/IP 关闭功能块
fbTcpClose(
	sSrvNetId:= ''   , 
	hSocket:=hTcpSock , 
	bExecute:=bClose , 
	tTimeout:=T#5S , 
	bBusy=> , 
	bError=> , 
	nErrId=> );


IF fbTcpCon.bBusy THEN
	bConnect:=FALSE;
END_IF

IF fbTcpClose.bBusy THEN
   bClose:=FALSE;
END_IF
END_ACTION

ACTION M_SendReceive:


  IF iCcd2.bSend THEN
	 bSendTcp:=TRUE;
	 iCcd2.bDone:=FALSE;
	 iCcd2.bError:=FALSE;
	 //iCcd2.strReceive:='';
    MEMSET(ADR(ccdDataSend.strBetryName),0,SIZEOF(ccdDataSend.strBetryName));
	MEMSET(ADR(ccdDataSend.strCode),0,SIZEOF(ccdDataSend.strCode));
	MEMSET(ADR(ccdDataSend.strShortData),0,SIZEOF(ccdDataSend.strShortData));
	MEMSET(ADR(ccdDataSend.strHotPress),0,SIZEOF(ccdDataSend.strHotPress));
    STRING_TO_UTF8(pDstUTF8:=ADR(ccdDataSend.strBetryName) , pSrcSTRING:=ADR(Data.strBetryName) , nDstSize:=INT_TO_UINT( LEN(STR:=Data.strBetryName )+1) );
    STRING_TO_UTF8(pDstUTF8:=ADR(ccdDataSend.strCode) , pSrcSTRING:=ADR(Data.strCode) , nDstSize:=INT_TO_UINT( LEN(STR:=Data.strCode )+1) ); 
    STRING_TO_UTF8(pDstUTF8:=ADR(ccdDataSend.strShortData) , pSrcSTRING:=ADR(Data.strShortData) , nDstSize:=INT_TO_UINT( LEN(STR:=Data.strShortData )+1) );
	STRING_TO_UTF8(pDstUTF8:=ADR(ccdDataSend.strHotPress) , pSrcSTRING:=ADR(Data.strHotPress) , nDstSize:=INT_TO_UINT( LEN(STR:=Data.strHotPress )+1) );
    iCcd2.bSend:=FALSE;
END_IF
	 

//第二步，编写 TCP/IP 发送功能块
fbTcpSend(
		sSrvNetId:= , 
		hSocket:=hTcpSock , //句柄；
		cbLen:=SIZEOF(ccdDataSend), //发送数据的长度；
		pSrc:= ADR(ccdDataSend), //发送数据指针的起始地址；
		bExecute:= bSendTcp, //发送执行位；
		tTimeout:= T#2S , 
		bBusy=> , 
		bError=> , 
		nErrId=> );
		
	IF bSendTcp AND fbTcpSend.bBusy THEN
		bSendTcp:=FALSE;
	END_IF
	
	
bReceiveTcp:=NOT bReceiveTcp;

//第三步，编写 TCP/IP 接收功能块
fbTcpRec(
	sSrvNetId:= , 
	hSocket:= hTcpSock, 
	cbLen:=SIZEOF(StrReceive) , //接收数据的长度；
	pDest:=ADR(StrReceive) , //接收数据指针的起始地址；
	bExecute:=bReceiveTcp , //接收执行位；
	tTimeout:= T#5S, 
	bBusy=> , 
	bError=> , 
	nErrId=> , 
	nRecBytes=> );

IF LEN(STR:=StrReceive )>=10 THEN
  iCcd2.strReceive:=StrReceive;
  StrReceive:='';
 // iCcd2.bDone:=TRUE;
END_IF


//IF LEN(STR:=StrReceive )=0 THEN
END_ACTION

END_FUNCTION_BLOCK

// ---- P2POUs/BasicFunction/12_User2/FB_CamDTDriver.TcPOU
FUNCTION_BLOCK FB_CamDTDriver	
VAR_INPUT
	Reset                                        :BOOL; //复位     
   	bCamInExecute			                :BOOL;	//凸轮耦合启动
   	bCreatTable		                        :BOOL;	//凸轮阶建启动
	iTable		                              :UINT;   //凸轮表号    
    fMainPos                                  :REAL;//叠台到位主轴的角度
    fbStartingPoint                           :REAL;//叠台凸轮的起点
	fbEndPoint								  :REAL;//叠台凸轮的终点
	fbCenterPoint								:REAL;//叠台压刀外边到过辊的中心距离
	
END_VAR
VAR_IN_OUT
	axisSlave		                    :axis_ref;  //从轴
	axisMaster		                    :axis_ref;  //主轴
	arrTableData: ARRAY[0..3600,0..1] OF LREAL;//叠台凸轮数据
END_VAR

VAR_OUTPUT
	Master_MidPos: LREAL;// 叠台压好到过辊中分主轴相位
	iFend: INT;// 叠台压刀到过辊中心主轴相位对应的索引	
    bCreatTableDone         :BOOL;//凸轮创建完成
    bCreatTableError         :BOOL;//凸轮创建错误
	bError                         :BOOL;//报警
	bReady                        :BOOL;//准备OK
	bInSync		                   :BOOL;//凸轮耦合中
END_VAR


VAR
	fbCamInSlave: MC_CamIn;
	fbCamOut: MC_CamOut;
	fbHaltSlave: MC_Halt; 
	rtrigs		:ARRAY[1..3]OF R_TRIG;
	ftrigs		:ARRAY[1..3]OF F_TRIG;
	iCamInStep: UINT;
	 PositionData			:	ARRAY[1..4] OF MC_MotionFunctionPoint;	
     PositionData1			:	ARRAY[1..4] OF MC_MotionFunctionPoint;	

	fbCamtableselect:			MC_CamTableSelect;
	Cam_table:				MC_CAM_REF;
    CamTable_MF:             MC_CAM_REF;

	rtError:  Tc2_Standard.R_TRIG;  	

    fbChangeCamModeSetOut	:	Tc2_MC2.ST_McOutputs;

	MA1: BOOL;
   fbCamInOut:                       Tc2_MC2.ST_McOutputs;
   bPoints :ARRAY[1..5] OF MC_MotionFunctionPoint; 
   mcReadMotionFunction: MC_ReadMotionFunction;
   mcReadMotionFunctionOut:Tc2_MC2.ST_McOutputs;
	iCreatTableStep: INT;
	fbHaltMaster: INT;
	bWriteCamData: BOOL;
	fSlavePos1: REAL;
	fSlavePos2: REAL;
	// 叠台移动的距离
	fBeltSpacePos: REAL;
	// 叠台中心点，主轴相位计算
	ReadPointVelues: BOOL;
	i: INT;
	Test_int: INT;
	mcReadMotionFunctionValues: MC_ReadMotionFunctionValues;
	CamTable: MC_CAM_REF;
	// 叠台凸轮数据读取完成
	arrReadPosDone: BOOL;
	rtRead: R_TRIG;
	ftRead: F_TRIG;	
	CamTable1: MC_CAM_REF;
	CamTable2: MC_CAM_REF;
	mcReadMotionFunctionValues_Busy: BOOL;
	mcReadMotionFunctionValues_Error: BOOL;
	mcReadMotionFunctionValues_ErrorID: UDINT;
	FB_ReadCamarrPos1: FB_ReadCamarrPos;
	arrReadPosDone1: BOOL;
	arrTableData1: ARRAY [0..3600, 0..1] OF LREAL;
	mcReadMotionFunctionValues1: MC_ReadMotionFunctionValues;
	CamTable3: MC_CAM_REF;
	TEST: BOOL;
END_VAR

rtrigs[1](CLK:=bCreatTable);  
ftrigs[1](CLK:=bCreatTable);  




CASE iCreatTableStep OF   
0:  
    IF  NOT bInSync  AND  rtrigs[1].Q  AND NOT bCreatTableError  THEN
         fbCamtableselect.Execute:=FALSE;
         bCreatTableDone:=FALSE;
         bCreatTable:=FALSE;
         bWriteCamData:=TRUE;
		 ReadPointVelues:=FALSE;
         iCreatTableStep:=10;
    END_IF 
10: //节点写入完成
   IF NOT bWriteCamData THEN 
	  fbCamtableselect.Execute:=TRUE;     
	 iCreatTableStep:=20;	
  END_IF
20:	//凸轮生成	
	IF NOT  fbCamtableselect.Execute     THEN
        //bCreatTableDone:=TRUE;
		iCreatTableStep:=30;	
    ELSIF  fbCamtableselect.Error THEN
       bCreatTableError:=TRUE;
       iCreatTableStep:=999;	//创建凸轮失败
	END_IF	
30:
		ReadPointVelues:=TRUE;
		IF arrReadPosDone THEN
			bCreatTableDone:=TRUE;
			ReadPointVelues:=FALSE;
			iCreatTableStep:=0;
		ELSIF mcReadMotionFunctionValues1.Error THEN
       		bCreatTableError:=TRUE;
       		iCreatTableStep:=999;	//创建凸轮失败			
		END_IF	
END_CASE	
(**********故障***********)
	IF  Reset  AND bCreatTableError  THEN  
	   bCreatTableError:=FALSE;
	   iCreatTableStep:=0;
	END_IF
(*****************************************耦合***************************************)
fbCamInSlave.BufferMode;
fbCamInSlave.Options.ActivationMode;
fbCamInSlave.Options.ActivationPosition;
fbCamInSlave.Options.ActivationMode;
fbCamInSlave.Options.InterpolationType;
fbCamInSlave.Options.MasterScalingMode;
fbCamInSlave.Options.SlaveScalingMode;

(************************************  相关状态  *************************************************)
bReady:= axisSlave.Status.ControlLoopClosed  AND axisMaster.Status.ControlLoopClosed AND  
               NOT bInSync  AND NOT bError   AND  bCreatTableDone   ;  

rtrigs[2](CLK:=bCamInExecute);  
ftrigs[2](CLK:=bCamInExecute);  

CASE iCamInStep OF
0:  
      fbCamInSlave.MasterOffset:=0;
      fbCamInSlave.SlaveOffset:=0;
      fbCamtableselect.Execute:=FALSE;
   	  fbCamInSlave.Execute:=FALSE;
	  fbCamOut.Execute:=FALSE;
	  fbHaltSlave.Execute:=FALSE;
      iCreatTableStep:=0;
      iCamInStep:=10;
10:
  IF bCamInExecute  AND  bReady THEN //耦合
	   iCamInStep:=100;
  ELSIF ftrigs[2].Q THEN  //解耦
	    iCamInStep:=200;
 ELSIF bInSync AND NOT bCamInExecute THEN
        iCamInStep:=200;
  END_IF

100:(**凸轮耦合**)
      fbCamInSlave.Execute:=TRUE;
      iCamInStep:=110;
110:
    IF NOT  fbCamInSlave.Execute AND axisSlave.Status.Coupled THEN
        bInSync:=TRUE;  //同步状态输出
        iCamInStep:=0;
   ELSIF fbCamInSlave.Error OR fbCamInSlave.CommandAborted THEN
         iCamInStep:=999;
    END_IF

(**********************解耦  *******************************)
200:
		fbCamOut.Execute:=TRUE;
		iCamInStep:=210;
210: 
	IF  NOT axisSlave.Status.Coupled   THEN 
	  	fbHaltSlave.Execute:=TRUE; 
	 	iCamInStep:=220;
    ELSIF  fbCamOut.Error  THEN
        iCamInStep:=999;
	END_IF
220: 
	IF axisSlave.Status.NotMoving    THEN
		bInSync:=FALSE; //同步状态输
		iCamInStep:=0;
     ELSIF fbHaltSlave.Error OR fbHaltSlave.CommandAborted THEN
          iCamInStep:=999;
	END_IF
END_CASE

(**********故障复位***********)
	IF  Reset  AND bError  THEN  
	   bError:=FALSE;
	   iCamInStep:=0;
	END_IF
rtError(CLK:=fbCamInSlave.Error  OR fbCamOut.Error OR fbHaltSlave.Error OR iCamInStep=999     , Q=> );
IF 	rtError.Q THEN
	bError:=TRUE;
	bInSync:=FALSE; //同步状态输
END_IF


Motion();      
ModifyCam();

ACTION ModifyCam:
//凸轮创建
fbCamtableselect(   
	Execute:=                        fbCamtableselect.Execute ,
	Periodic:=                       TRUE ,
	MasterAbsolute:=             FALSE,//
	SlaveAbsolute:=                FALSE ,//
	CamTableID:=                  iTable,
	Master:=                         axisMaster ,
	Slave:=                            axisSlave ,
	CamTable:=                     Cam_table , );
IF fbCamtableselect.Done THEN
    fbCamtableselect.Execute:=FALSE;
END_IF
//凸轮关键点写入
IF bWriteCamData  THEN    //98     初始点   90
	  Cam_table.ArraySize:=SIZEOF(PositionData1); 
	  Cam_table.NoOfColumns:=1;
	  Cam_table.NoOfRows:=3;
	  Cam_table.pArray:=ADR(PositionData1);
	  Cam_table.TableType:=MC_TABLETYPE_MOTIONFUNCTION;
  
	  fBeltSpacePos:=fbEndPoint-fbStartingPoint;
	  
	  PositionData1[1].	PointIndex	:=	        1;
	  PositionData1[1].	FunctionType	:=		MOTIONFUNCTYPE_POLYNOM7_MM;
	  PositionData1[1].	PointType	:=	        MOTIONPOINTTYPE_MOTION;
	  PositionData1[1].	RelIndexNextPoint	:=  1;
	  PositionData1[1].	MasterPos	:=	        0;
	  PositionData1[1].	SlavePos	:=	        0;		
	  PositionData1[1].	SlaveVelo	:=	        0;
	  
	  PositionData1[2].	PointIndex	:=	        2;
	  PositionData1[2].	FunctionType	:=		MOTIONFUNCTYPE_POLYNOM1;
	  PositionData1[2].	PointType	:=	        MOTIONPOINTTYPE_MOTION;
	  PositionData1[2].	RelIndexNextPoint	:=  1;
	  PositionData1[2].	MasterPos	:=	        fMainPos;
	  PositionData1[2].	SlavePos	:=	        fBeltSpacePos;	
	  PositionData1[2].	SlaveVelo	:=	        0	;
	  
	  PositionData1[3].	PointIndex	:=	        3;
	  PositionData1[3].	FunctionType	:=		MOTIONFUNCTYPE_POLYNOM7_MM;
	  PositionData1[3].	PointType	:=	        MOTIONPOINTTYPE_MOTION;
	  PositionData1[3].	RelIndexNextPoint	:=  0;
	  PositionData1[3].	MasterPos	:=	        360;
	  PositionData1[3].	SlavePos	:=	        fBeltSpacePos;	
	  PositionData1[3].	SlaveVelo	:=	       0;
   
     bWriteCamData:=FALSE;
END_IF


